// TIA Portal project "DT_PSA_OPCV" (V19)

(* hardware
DEVICE "S7-1500/ET200MP-Station_1"  S7-1500 station
   slot 0: "Profilschiene_0"  Rack  6ES7 590-1***0-0AA0
   slot 1: "PLC_1"  CPU 1516F-3 PN/DP  6ES7 516-3FN02-0AB0  V2.9
      slot 3: "CPU-Display_1"  6ES7591-1BA00-0AA0
      slot 32768: "PROFINET-Schnittstelle_1"  X1
         slot 32769: "Port_1"  X1 P1
         slot 32770: "Port_2"  X1 P2
      slot 33024: "PROFINET-Schnittstelle_2"  X2
         slot 33025: "Port_1"  X2 P1
      slot 33280: "DP-Schnittstelle_1"  X3
      slot 34817: "Virtual CP interface port_1"  Virtual CP interface port  Virtual CP interface port
   slot 2: "DI 16x24VDC HF_1"  DI 16x24VDC HF  6ES7 521-1BH00-0AB0  V2.2
   slot 3: "DQ 8x24VDC/2A HF_1"  DQ 8x24VDC/2A HF  6ES7 522-1BF00-0AB0  V2.2
   slot 4: "F-DI 16x24V DC_1"  F-DI 16x24V DC  6ES7 526-1BH00-0AB0  V1.0
      slot 1: "F-DI 16x24V DC_1"  F-DI 16x24V DC
   slot 5: "F-DQ 8x24V DC/2A PPM_1"  F-DQ 8x24V DC/2A PPM  6ES7 526-2BF00-0AB0  V1.0
      slot 1: "F-DQ 8x24V DC/2A PPM_1"  F-DQ 8x24V DC/2A PPM
DEVICE "HMI_1"  TP700 Comfort
   slot 0: "HMI_1"  TP700 Comfort  6AV2 124-0GC01-0AX0  17.0.0.0
   slot 1: "HMI_RT_1"  TP700 Comfort  6AV2 124-0GC01-0AX0  17.0.0.0
   slot 5: "HMI_1.IE_CP_1"  PROFINET Interface  17.0.0.0
      slot 1: "PROFINET Schnittstelle_1"  PROFINET Interface
         slot 1: "Port_1"  Port
         slot 2: "Port_2"  Port
   slot 7: "HMI_1.MPI/DP_CP_1"  MPI/DP Interface  17.0.0.0
*)

// ===== PLC "PLC_1"  CPU 1516F-3 PN/DP =====
// protected blocks, not shown: "Main_Safety_RTG1", "Main_Safety_RTG1_DB"

VAR_GLOBAL   // PLC tag table "Control Panel"
   "BT2_OpMode" AT %I0.2 : Bool;   // Betriebsart: 1=Automatik / 0=Hand
   "BT3_SingleStep" AT %I0.3 : Bool;   // Einzelschritt ausführen
   "BT4_AutoStart" AT %I0.4 : Bool;   // Automatik Ein
   "BT5_AutoStop" AT %I0.5 : Bool;   // Automatik Halt
   "BT7_Reset" AT %I0.7 : Bool;   // Grundstellung
   "BT6_Ack" AT %I0.6 : Bool;   // Störung quittieren
   "BT1_ControlLight" AT %Q0.1 : Bool;   // Tasterbeleuchtung "Steuerung läuft" (grün)
   "BT4_AutoLight" AT %Q0.4 : Bool;   // Tasterbeleuchtung "Automatik läuft" (grün)
   "BT6_ErrFltLight" AT %Q0.6 : Bool;   // Tasterbeleuchtung "Lampe Störung" (rot)
   "SignalTower_Yellow" AT %Q1.2 : Bool;   // Ampel "Lampe Einrichten aktiv" (gelb)
   "BT1_ControlOnOff" AT %I0.1 : Bool;   // 1 = Steuerung Ein (einrastend)
   "SignalTower_Green" AT %Q1.1 : Bool;   // Ampel "Automatik läuft" (grün)
   "SignalTower_Red" AT %Q1.3 : Bool;   // Ampel "Störung" (rot)
   "BT3_SingleStepLight" AT %Q0.3 : Bool;   // Tasterbeleuchtung "Einzelschritt läuft" (grün)
   "BT7_HomingLight" AT %Q0.7 : Bool;   // Tasterbeleuchtung "Grundstellungsfahrt läuft" (green)
   "BT5_AutoStopLight" AT %Q0.5 : Bool;   // Tasterbeleuchtung "Automatik Stop läuft" (blau)
   "BT8_ImmediateStop" AT %I1.0 : Bool;   // Sofort Halt
   "BT8_ImmediateStopLight" AT %Q1.0 : Bool;   // Tasterbeleuchtung "Sofort Halt" (rot)
END_VAR

VAR_GLOBAL   // PLC tag table "System"
   "Clock_Byte" AT %MB0 : Byte;
   "Clock_10Hz" AT %M0.0 : Bool;
   "Clock_5Hz" AT %M0.1 : Bool;
   "Clock_2.5Hz" AT %M0.2 : Bool;
   "Clock_2Hz" AT %M0.3 : Bool;
   "Clock_1.25Hz" AT %M0.4 : Bool;
   "Clock_1Hz" AT %M0.5 : Bool;
   "Clock_0.625Hz" AT %M0.6 : Bool;
   "Clock_0.5Hz" AT %M0.7 : Bool;
   "System_Byte" AT %MB1 : Byte;
   "FirstScan" AT %M1.0 : Bool;
   "DiagStatusUpdate" AT %M1.1 : Bool;
   "AlwaysTRUE" AT %M1.2 : Bool;
   "AlwaysFALSE" AT %M1.3 : Bool;
   "Commissioning_True" AT %M2.0 : Bool;
END_VAR

VAR_GLOBAL CONSTANT   // PLC tag table "System"
   "SYS_MACHINE_MAXSTATIONS" : USInt := 10;   // Anzahl Stationen pro Maschine
   "SYS_SQ_MAXSEQUENCES" : USInt := 12;   // Anzahl Schrittketten pro Station
   "SYS_DRIVE_POSITIONS" : USInt := 8;   // Anzahl Positionen pro Servoantrieb
   "SYS_MANUALMOVEMENTS" : UInt := 64;   // Anzahl maximaler Einrichtfunktionen
   "SYS_HMI_SETUPMAXROWS" : USInt := 6;   // HMI Vorgabe maximale Anzahl an Einrichtzeilen auf der Steuerung verfügbar
END_VAR

VAR_GLOBAL   // PLC tag table "FG01"
   "FG01_Y_Gripper_InHome" AT %I101.0 : Bool;   // geöffnet
   "FG01_Y_Gripper_InWork" AT %I101.1 : Bool;   // geschlossen
   "FG01_Y_Gripper_WorkPos" AT %Q101.1 : Bool;   // schließen
   "FG01_Y_Plattform_InHome" AT %I102.0 : Bool;   // hinten
   "FG01_Y_Plattform_InWork" AT %I102.1 : Bool;   // vorne
   "FG01_Y_Plattform_HomePos" AT %Q102.0 : Bool;
   "FG01_Y_Plattform_WorkPos" AT %Q102.1 : Bool;
   "FG01_Y_ReaderWindow_InWork" AT %I103.1 : Bool;
   "FG01_Y_ReaderWindow_WorkPos" AT %Q103.1 : Bool;   // Position zum Code Lesen
   "FG01_Y_Gripper_HomePos" AT %Q101.0 : Bool;   // öffnen
   "FG01_Y_ReaderWindow_HomePos" AT %Q103.0 : Bool;
END_VAR

VAR_GLOBAL   // PLC tag table "FG03"
   "FG03_Y_AxisR1_InHome" AT %I301.0 : Bool;
   "FG03_Y_AxisR1_InWork" AT %I301.1 : Bool;
   "FG03_Y_AxisR1_HomePos" AT %Q301.0 : Bool;
   "FG03_Y_AxisR1_WorkPos" AT %Q301.1 : Bool;
   "FG03_Y_AxisX1_InHome" AT %I302.0 : Bool;
   "FG03_Y_AxisX1_InWork" AT %I302.1 : Bool;
   "FG03_Y_AxisX1_HomePos" AT %Q302.0 : Bool;
   "FG03_Y_AxisX1_WorkPos" AT %Q302.1 : Bool;
   "FG03_Y_AxisY1_InHome" AT %I303.0 : Bool;
   "FG03_Y_AxisY1_InWork" AT %I303.1 : Bool;
   "FG03_Y_AxisY1_HomePos" AT %Q303.0 : Bool;
   "FG03_Y_AxisY1_WorkPos" AT %Q303.1 : Bool;
   "FG03_Y_AxisX2_InHome" AT %I304.0 : Bool;
   "FG03_Y_AxisX2_InWork" AT %I304.1 : Bool;
   "FG03_Y_AxisX2_HomePos" AT %Q304.0 : Bool;
   "FG03_Y_AxisX2_WorkPos" AT %Q304.1 : Bool;
   "FG03_Y_AxisY2_InHome" AT %I305.0 : Bool;
   "FG03_Y_AxisY2_InWork" AT %I305.1 : Bool;
   "FG03_Y_AxisY2_HomePos" AT %Q305.0 : Bool;
   "FG03_Y_AxisY2_WorkPos" AT %Q305.1 : Bool;
   "FG03_Y_Gripper1_InHome" AT %I306.0 : Bool;
   "FG03_Y_Gripper1_InWork" AT %I306.1 : Bool;
   "FG03_Y_Gripper1_HomePos" AT %Q306.0 : Bool;
   "FG03_Y_Gripper1_WorkPos" AT %Q306.1 : Bool;
   "FG03_Y_Gripper2_InHome" AT %I307.0 : Bool;
   "FG03_Y_Gripper2_InWork" AT %I307.1 : Bool;
   "FG03_Y_Gripper2_HomePos" AT %Q307.0 : Bool;
   "FG03_Y_Gripper2_WorkPos" AT %Q307.1 : Bool;
END_VAR

VAR_GLOBAL   // PLC tag table "FG04"
   "FG04_Y_AxisZ_InWork" AT %I401.1 : Bool;
   "FG04_Y_AxisZ_WorkPos" AT %Q401.1 : Bool;
   "FG04_Y_AxisZ_HomePos" AT %Q401.0 : Bool;
   "FG04_Y_AxisZ_InHome" AT %I401.0 : Bool;
END_VAR

VAR_GLOBAL   // PLC tag table "FG05"
   "FG05_B_Part" AT %I500.0 : Bool;
   "FG05_Y_AxisR_InHome" AT %I501.0 : Bool;
   "FG05_Y_AxisR_InWork" AT %I501.1 : Bool;
   "FG05_Y_AxisR_HomePos" AT %Q501.0 : Bool;
   "FG05_Y_AxisR_WorkPos" AT %Q501.1 : Bool;
   "FG05_Y_AxisX_InHome" AT %I502.0 : Bool;
   "FG05_Y_AxisX_InWork" AT %I502.1 : Bool;
   "FG05_Y_AxisX_HomePos" AT %Q502.0 : Bool;
   "FG05_Y_AxisX_WorkPos" AT %Q502.1 : Bool;
   "FG05_Y_AxisZ1_InHome" AT %I503.0 : Bool;
   "FG05_Y_AxisZ1_InWork" AT %I503.1 : Bool;
   "FG05_Y_AxisZ1_HomePos" AT %Q503.0 : Bool;
   "FG05_Y_AxisZ1_WorkPos" AT %Q503.1 : Bool;
   "FG05_Y_AxisZ2_InHome" AT %I504.0 : Bool;
   "FG05_Y_AxisZ2_InWork" AT %I504.1 : Bool;
   "FG05_Y_AxisZ2_HomePos" AT %Q504.0 : Bool;
   "FG05_Y_AxisZ2_WorkPos" AT %Q504.1 : Bool;
   "FG05_Y_CapsSourceStopper_InHome" AT %I505.0 : Bool;   // GS = Kaps können vereinzelt werden
   "FG05_Y_CapsSourceStopper_WorkPos" AT %Q505.1 : Bool;   // AS = Vereinzelung kann geleert werden (Vereinzelung nicht möglich)
   "FG05_Y_Gripper_InHome" AT %I506.0 : Bool;
   "FG05_Y_Gripper_InWork" AT %I506.1 : Bool;
   "FG05_Y_Gripper_HomePos" AT %Q506.0 : Bool;
   "FG05_Y_Gripper_WorkPos" AT %Q506.1 : Bool;
   "FG05_Y_CapsSourceStopper_HomePos" AT %Q505.0 : Bool;
   "FG05_M_Bunker" AT %Q507.0 : Bool;   // Sortiertopf ein
   "FG05_M_Conveyor" AT %Q507.1 : Bool;   // Linearförderer ein
END_VAR

VAR_GLOBAL   // PLC tag table "FG_Transport"
   "FG_TS_Gate_1_InHome" AT %I1001.0 : Bool;   // geöffnet
   "FG_TS_Gate_1_InWork" AT %I1001.1 : Bool;   // geschlossen
   "FG_TS_Gate_1_WorkPos" AT %Q1001.1 : Bool;   // Schließen
   "FG_TS_Gate_2_InHome" AT %I1002.0 : Bool;   // geöffnet
   "FG_TS_Gate_2_InWork" AT %I1002.1 : Bool;   // geschlossen
   "FG_TS_Gate_2_WorkPos" AT %Q1002.1 : Bool;   // Schließen
   "FG_TS_Index01_B_Detect" AT %I1003.0 : Bool;   // 1 = erkannt
   "FG_TS_Index01_B_Exit" AT %I1003.1 : Bool;   // 1 = erkannt
   "FG_TS_Index01_Y_Lift_InHome" AT %I1003.2 : Bool;   // Heber ist unten
   "FG_TS_Index01_Y_Lift_InWork" AT %I1003.3 : Bool;   // Heber ist oben
   "FG_TS_Index01_Y_Lift_HomePos" AT %Q1003.0 : Bool;   // Heber senken
   "FG_TS_Index01_Y_Lift_WorkPos" AT %Q1003.1 : Bool;   // Heber heben
   "FG_TS_Index01_Y_Stopper_InHome" AT %I1003.4 : Bool;   // Stopper geschlossen
   "FG_TS_Index01_Y_Stopper_WorkPos" AT %Q1003.2 : Bool;   // Stopper öffnen
   "FG_TS_Index02_B_Detect" AT %I1004.0 : Bool;   // 1 = erkannt
   "FG_TS_Index02_B_Exit" AT %I1004.1 : Bool;   // 1 = erkannt
   "FG_TS_Index02_Y_Lift_InHome" AT %I1004.2 : Bool;   // Heber ist unten
   "FG_TS_Index02_Y_Lift_InWork" AT %I1004.3 : Bool;   // Heber ist oben
   "FG_TS_Index02_Y_Lift_HomePos" AT %Q1004.0 : Bool;   // Heber senken
   "FG_TS_Index02_Y_Lift_WorkPos" AT %Q1004.1 : Bool;   // Heber heben
   "FG_TS_Index02_Y_Stopper_InHome" AT %I1004.4 : Bool;   // Stopper geschlossen
   "FG_TS_Index02_Y_Stopper_WorkPos" AT %Q1004.2 : Bool;   // Stopper öffnen
   "FG_TS_Index03_B_Detect" AT %I1005.0 : Bool;   // 1 = erkannt
   "FG_TS_Index03_B_Exit" AT %I1005.1 : Bool;   // 1 = erkannt
   "FG_TS_Index03_Y_Lift_InHome" AT %I1005.2 : Bool;   // Heber ist unten
   "FG_TS_Index03_Y_Lift_InWork" AT %I1005.3 : Bool;   // Heber ist oben
   "FG_TS_Index03_Y_Lift_HomePos" AT %Q1005.0 : Bool;   // Heber senken
   "FG_TS_Index03_Y_Lift_WorkPos" AT %Q1005.1 : Bool;   // Heber heben
   "FG_TS_Index03_Y_Stopper_InHome" AT %I1005.4 : Bool;   // Stopper geschlossen
   "FG_TS_Index03_Y_Stopper_WorkPos" AT %Q1005.2 : Bool;   // Stopper öffnen
   "FG_TS_Index04_B_Detect" AT %I1006.0 : Bool;   // 1 = erkannt
   "FG_TS_Index04_B_Exit" AT %I1006.1 : Bool;   // 1 = erkannt
   "FG_TS_Index04_Y_Lift_InHome" AT %I1006.2 : Bool;   // Heber ist unten
   "FG_TS_Index04_Y_Lift_InWork" AT %I1006.3 : Bool;   // Heber ist oben
   "FG_TS_Index04_Y_Lift_HomePos" AT %Q1006.0 : Bool;   // Heber senken
   "FG_TS_Index04_Y_Lift_WorkPos" AT %Q1006.1 : Bool;   // Heber heben
   "FG_TS_Index04_Y_Stopper_InHome" AT %I1006.4 : Bool;   // Stopper geschlossen
   "FG_TS_Index04_Y_Stopper_WorkPos" AT %Q1006.2 : Bool;   // Stopper öffnen
   "FG_TS_Index05_B_Detect" AT %I1007.0 : Bool;   // 1 = erkannt
   "FG_TS_Index05_B_Exit" AT %I1007.1 : Bool;   // 1 = erkannt
   "FG_TS_Index05_Y_Lift_InHome" AT %I1007.2 : Bool;   // Heber ist unten
   "FG_TS_Index05_Y_Lift_InWork" AT %I1007.3 : Bool;   // Heber ist oben
   "FG_TS_Index05_Y_Lift_HomePos" AT %Q1007.0 : Bool;   // Heber senken
   "FG_TS_Index05_Y_Lift_WorkPos" AT %Q1007.1 : Bool;   // Heber heben
   "FG_TS_Index05_Y_Stopper_InHome" AT %I1007.4 : Bool;   // Stopper geschlossen
   "FG_TS_Index05_Y_Stopper_WorkPos" AT %Q1007.2 : Bool;   // Stopper öffnen
   "FG_TS_Stopper01_B_Detect" AT %I1008.0 : Bool;   // 1 = erkannt
   "FG_TS_Stopper01_B_Exit" AT %I1008.1 : Bool;   // 1 = erkannt
   "FG_TS_Stopper01_Y_Stopper_InHome" AT %I1008.4 : Bool;   // Stopper geschlossen
   "FG_TS_Stopper01_Y_Stopper_WorkPos" AT %Q1008.2 : Bool;   // Stopper öffnen
   "FG_TS_Stopper02_B_Detect" AT %I1009.0 : Bool;   // 1 = erkannt
   "FG_TS_Stopper02_B_Exit" AT %I1009.1 : Bool;   // 1 = erkannt
   "FG_TS_Stopper02_Y_Stopper_InHome" AT %I1009.4 : Bool;   // Stopper geschlossen
   "FG_TS_Stopper02_Y_Stopper_WorkPos" AT %Q1009.2 : Bool;   // Stopper öffnen
   "FG_TS_Stopper03_B_Detect" AT %I1010.0 : Bool;   // 1 = erkannt
   "FG_TS_Stopper03_B_Exit" AT %I1010.1 : Bool;   // 1 = erkannt
   "FG_TS_Stopper03_Y_Stopper_InHome" AT %I1010.4 : Bool;   // Stopper geschlossen
   "FG_TS_Stopper03_Y_Stopper_WorkPos" AT %Q1010.2 : Bool;   // Stopper öffnen
   "FG_TS_Stopper04_B_Detect" AT %I1011.0 : Bool;   // 1 = erkannt
   "FG_TS_Stopper04_B_Exit" AT %I1011.1 : Bool;   // 1 = erkannt
   "FG_TS_Stopper04_Y_Stopper_InHome" AT %I1011.4 : Bool;   // Stopper geschlossen
   "FG_TS_Stopper04_Y_Stopper_WorkPos" AT %Q1011.2 : Bool;   // Stopper öffnen
   "FG_TS_Lift01_B_Detect" AT %I1012.0 : Bool;   // 1 = erkannt
   "FG_TS_Lift01_B_Exit" AT %I1012.1 : Bool;   // 1 = erkannt
   "FG_TS_Lift01_Y_Lift_InHome" AT %I1012.2 : Bool;   // Heber ist unten
   "FG_TS_Lift01_Y_Lift_InWork" AT %I1012.3 : Bool;   // Heber ist oben
   "FG_TS_Lift01_Y_Lift_HomePos" AT %Q1012.0 : Bool;   // Heber senken
   "FG_TS_Lift01_Y_Lift_WorkPos" AT %Q1012.1 : Bool;   // Heber heben
   "FG_TS_Lift01_M_Conveyor_Plus" AT %Q1012.2 : Bool;   // Antrieb vorwärts
   "FG_TS_Lift01_M_Conveyor_Minus" AT %Q1012.3 : Bool;   // Antrieb rückwärts
   "FG_TS_Lift02_B_Detect" AT %I1013.0 : Bool;   // 1 = erkannt
   "FG_TS_Lift02_B_Exit" AT %I1013.1 : Bool;   // 1 = erkannt
   "FG_TS_Lift02_Y_Lift_InHome" AT %I1013.2 : Bool;   // Heber ist unten
   "FG_TS_Lift02_Y_Lift_InWork" AT %I1013.3 : Bool;   // Heber ist oben
   "FG_TS_Lift02_Y_Lift_HomePos" AT %Q1013.0 : Bool;   // Heber senken
   "FG_TS_Lift02_Y_Lift_WorkPos" AT %Q1013.1 : Bool;   // Heber heben
   "FG_TS_Lift02_M_Conveyor_Plus" AT %Q1013.2 : Bool;   // Antrieb vorwärts
   "FG_TS_Lift02_M_Conveyor_Minus" AT %Q1013.3 : Bool;   // Antrieb rückwärts
   "FG_TS_Transport01_M_Conveyor_Plus" AT %Q1014.0 : Bool;   // Antrieb vorwärts
   "FG_TS_Transport01_M_Conveyor_Minus" AT %Q1014.1 : Bool;   // Antrieb rückwärts
   "FG_TS_Transport02_M_Conveyor_Plus" AT %Q1015.0 : Bool;   // Antrieb vorwärts
   "FG_TS_Transport02_M_Conveyor_Minus" AT %Q1015.1 : Bool;   // Antrieb rückwärts
END_VAR

VAR_GLOBAL   // PLC tag table "Safety"
   "i_SS_ESTOP1" AT %I50.0 : Bool;
   "q_SS_ESTOP1" AT %Q50.0 : Bool;
END_VAR

// folder: Actors/ActorTypes

TYPE "typeActor"
   STRUCT
      setHomePos : Bool;   // Grundstellung ansteuern
      setWorkPos : Bool;   // Arbeitsstellung ansteuern
      inHomePos : Bool;   // steht in Grundstellung
      inWorkPos : Bool;   // steht in Arbeitsstellung
      homeAct : Bool;   // Grundstellung wird angesteuert
      workAct : Bool;   // Arbeitsstellung wird angesteuert
      homeIsInterlocked : Bool;   // 1 = Grundstellung ist gesperrt
      workIsInterlocked : Bool;   // 1 = Arbeitsstellung ist gesperrt
   END_STRUCT;
END_TYPE

TYPE "typeActor_2Out0In"
   STRUCT
      setHomePos : Bool;   // Grundstellung ansteuern
      setWorkPos : Bool;   // Arbeitsstellung ansteuern
      homeAct : Bool;   // Grundstellung wird angesteuert
      workAct : Bool;   // Arbeitsstellung wird angesteuert
      homeIsInterlocked : Bool;   // 1 = Grundstellung ist gesperrt
      workIsInterlocked : Bool;   // 1 = Arbeitsstellung ist gesperrt
      setError : Bool;   // in Störung setzen
      inError : Bool;   // Störung vorhanden
   END_STRUCT;
END_TYPE

TYPE "typeActor_2Out2In"
   STRUCT
      setHomePos : Bool;   // Grundstellung ansteuern
      setWorkPos : Bool;   // Arbeitsstellung ansteuern
      inHomePos : Bool;   // steht in Grundstellung
      inWorkPos : Bool;   // steht in Arbeitsstellung
      homeAct : Bool;   // Grundstellung wird angesteuert
      workAct : Bool;   // Arbeitsstellung wird angesteuert
      homeIsInterlocked : Bool;   // 1 = Grundstellung ist gesperrt
      workIsInterlocked : Bool;   // 1 = Arbeitsstellung ist gesperrt
      setError : Bool;   // in Störung setzen
      inError : Bool;   // Störung vorhanden
   END_STRUCT;
END_TYPE

TYPE "typeActor_1Out0In"
   STRUCT
      setWorkPos : Bool;   // Arbeitsstellung ansteuern
      workAct : Bool;   // Arbeitsstellung wird angesteuert
      workIsInterlocked : Bool;   // 1 = Arbeitsstellung ist gesperrt
      setError : Bool;   // in Störung setzen
      inError : Bool;   // Störung vorhanden
   END_STRUCT;
END_TYPE

TYPE "typeActor_1Out2In"
   STRUCT
      setWorkPos : Bool;   // Arbeitsstellung ansteuern
      inHomePos : Bool;   // steht in Grundstellung
      inWorkPos : Bool;   // steht in Arbeitsstellung
      workAct : Bool;   // Arbeitsstellung wird angesteuert
      workIsInterlocked : Bool;   // 1 = Arbeitsstellung ist gesperrt
      setError : Bool;   // in Störung setzen
      inError : Bool;   // Störung vorhanden
   END_STRUCT;
END_TYPE

TYPE "typeActor_2Out1In"
   STRUCT
      setHomePos : Bool;   // Grundstellung ansteuern
      setWorkPos : Bool;   // Arbeitsstellung ansteuern
      inHomePos : Bool;   // steht in Grundstellung
      inWorkPos : Bool;   // steht in Arbeitsstellung
      homeAct : Bool;   // Grundstellung wird angesteuert
      workAct : Bool;   // Arbeitsstellung wird angesteuert
      homeIsInterlocked : Bool;   // 1 = Grundstellung ist gesperrt
      workIsInterlocked : Bool;   // 1 = Arbeitsstellung ist gesperrt
      setError : Bool;   // in Störung setzen
      inError : Bool;   // Störung vorhanden
   END_STRUCT;
END_TYPE

TYPE "typeActor_1Out1In"
   STRUCT
      setWorkPos : Bool;   // Arbeitsstellung ansteuern
      inHomePos : Bool;   // steht in Grundstellung
      inWorkPos : Bool;   // steht in Arbeitsstellung
      workAct : Bool;   // Arbeitsstellung wird angesteuert
      workIsInterlocked : Bool;   // 1 = Arbeitsstellung ist gesperrt
      setError : Bool;   // in Störung setzen
      inError : Bool;   // Störung vorhanden
   END_STRUCT;
END_TYPE

// folder: Actors/Drives

TYPE "typeDriveData"
   STRUCT
      position : Array[1.."SYS_DRIVE_POSITIONS"] of Real;   // Positionsvorgabe
      speed : Array[1.."SYS_DRIVE_POSITIONS"] of Real;   // Geschwindigkeitsvorgabe
   END_STRUCT;
   // // position[1] : Grundstellung (reserviert)
END_TYPE

TYPE "typeDriveControl"
   STRUCT
      moveToPos : Array[1.."SYS_DRIVE_POSITIONS"] of Bool;   // Fahrbefehl ausführen
      jog : Struct   // Handbetrieb
         pos : Bool;   // Tippen positiv
         neg : Bool;   // Tippen negativ
         "step" : Real;   // Tippschrittweite
         speed : Real;   // Tippgeschwindigkeit
      END_STRUCT;
   END_STRUCT;
END_TYPE

TYPE "typeDriveStatus"
   STRUCT
      ready : Bool;   // Bereit
      error : Bool;   // Störung
      posReached : Bool;   // Positionsvorgabe erreicht
      actualPosition : Real;   // Ist-Position
      actualSpeed : Real;   // Ist-Geschwindigkeit
      interlockMin : Bool;   // 1 = Fahrtrichtung zur Endposition min gesperrt
      interlockMax : Bool;   // 1 = Fahrtrichtung zur Endposition max gesperrt
      endPosMin : Bool;   // Endposition min erreicht
      endPosMax : Bool;   // Endposition max erreicht
      inHomePos : Bool;   // steht in Grundstellung
   END_STRUCT;
END_TYPE

TYPE "typeDriveConverter"
   STRUCT
      actualPosition : Real;   // Ist-Position (Drive-Einheit)
      actualSpeed : Real;   // Ist-Geschwindigkeit (Drive-Einheit)
      setPosition : Real;   // Sollposition (Drive-Einheit)
      setSpeed : Real;   // Sollgeschwindigkeit (Drive-Einheit)
      minPosDrive : Real;   // Minimale Positionierung (Drive-Einheit)
      maxPosDrive : Real;   // Maximale Positionierung (Drive-Einheit)
      maxSpeedDrive : Real;   // Maximale Geschwindigkeit (Drive-Einheit)
      posOffset : Real;   // Offset für Positionsfensterfreigabe (Drive-Einheit)
      ready : Bool;   // Umrichter Bereit
      error : Bool;   // Umrichter Störung
      posReached : Bool;   // Position erreicht
      releaseMotion : Bool;   // Bewegungsfreigabe
   END_STRUCT;
END_TYPE

// folder: HMI/Errors_Messages

TYPE "typePlcErrors"
   STRUCT
      errorNo : Array[1..64] of Bool;
   END_STRUCT;
END_TYPE

TYPE "typeHmiErrMsg"
   STRUCT
      message : Array[1..2] of Word;   // Meldung auslösen
      alarmAckPlc : Array[1..8] of Word;   // Fehler auslösen und Quittierung über SPS
      ackHmi : Array[1..4] of Word;   // Quittierung über HMI
   END_STRUCT;
END_TYPE

TYPE "typePlcErrMsg"
   STRUCT
      messages : "typePlcMessages";
      alarms : "typePlcErrors";
   END_STRUCT;
END_TYPE

TYPE "typePlcMessages"
   STRUCT
      msgNo : Array[1..32] of Bool;
   END_STRUCT;
END_TYPE

// folder: HMI/ManualMovement

TYPE "typeHmiManualMove"
   STRUCT
      move : "typeManualMove";   // Bewegung
      movementNo : USInt;   // Nummer der Bewegungsfunktion
      textlistFunctionName : UInt;   // Funktionsname: Wert für Textliste
      textlistFunctionExecuteLeft : UInt;   // Bewegung Links: Wert für Textliste
      textlistFunctionFinalPosLeft : UInt;   // Endposition Links: Wert für Textliste
      textlistFunctionExecuteRight : UInt;   // Bewegung Rechts: Wert für Textliste
      textlistFunctionFinalPosRight : UInt;   // Endposition Rechts: Wert für Textliste
   END_STRUCT;
END_TYPE

TYPE "typeHmiManualMovement"
   STRUCT
      selection : Struct
         station : USInt;   // Angewählte Station
         page : USInt;   // Aktuele Seite
         ofMaxPages : USInt;   // von maximal Seiten
         nextPage : Bool;   // Schaltfläche: Nächste Seite
         previousPage : Bool;   // Schaltfläche: Vorherige Seite
         showSymbols : Bool;   // Schaltfläche: Zeige symbolische Ansicht
      END_STRUCT;
      rows : Array[1.."SYS_HMI_SETUPMAXROWS"] of "typeHmiManualMove";
   END_STRUCT;
END_TYPE

// folder: Machine

TYPE "typeMachine"
   STRUCT
      controlOn : Bool;   // Maschinensteuerung ist eingeschaltet
      automaticMode : Bool;   // Betriebsart Automatik ist aktiv
      automaticIsRunning : Bool;   // Automatik (bzw. ReleaseCycle) läuft in mindestens einer Station
      automaticStart : Bool;   // Automatikstart auslösen
      automaticStops : Bool;   // Automatik stoppt
      singleStepPulse : Bool;   // Einzelschritt
      immediateStop : Bool;   // Sofort Halt der Stationen auslösen
      acknowledge : Bool;   // Quittierung
      reset : Bool;   // Neustart/Grundstellung auslösen
      isInError : Bool;   // Störung vorhanden
      isHoming : Bool;   // Maschinengrundstellungsfahrt wird ausgeführt
      isInHome : Bool;   // Alle Stationen sind in Grundstellung
   END_STRUCT;
END_TYPE

TYPE "typeStation"
   STRUCT
      exists : Bool := false;   // true = Station existiert / false = Platzhalter
      signals : "typeStationSignals";
      stepSeqs : "typeStepSequences";
   END_STRUCT;
END_TYPE

TYPE "typeStations"
   STRUCT
      station : Array[1.."SYS_MACHINE_MAXSTATIONS"] of "typeStation";
   END_STRUCT;
END_TYPE

TYPE "typeStepSequence"
   STRUCT
      exists : Bool;   // Schrittkette verfügbar
      start : Bool;   // Start Schrittkette
      running : Bool;   // Schrittkette läuft
      done : Bool;   // Schrittkette ist fertig
      error : Bool;   // Störung vorhanden
      init : Bool;   // Initialschritt aktiv
      inHome : Bool;   // Steht in Grundstellung
      isWaiting : Bool;   // Steht im Warteschritt
      inHoming : Bool;   // Grundstellungsfahrt aktiv
      jogDone : Bool;   // Halbautomatische Weiterschaltung abgeschlossen
   END_STRUCT;
END_TYPE

TYPE "typeStepSequences"
   STRUCT
      stepSeq : Array[1.."SYS_SQ_MAXSEQUENCES"] of "typeStepSequence";   // Schrittkette
   END_STRUCT;
END_TYPE

TYPE "typeMachineSafety"
   STRUCT
      EStopOk : Bool;   // Not-Aus Kreis ok
      RunUpPneumatic : Bool;
      PneumaticIsOk : Bool;
      Error : Bool;
   END_STRUCT;
END_TYPE

TYPE "typeStationSignals"
   STRUCT
      safetyOk : Bool;   // Sicherheit ist ok
      controlOn : Bool;   // Steuerung eingeschaltet
      automaticMode : Bool;   // Automatikmodus angewählt
      modeSetup : Bool;   // Handmodus angewählt
      modeAuto : Bool;   // Betriebsart: Automatik aktiv
      modeTap : Bool;   // Betriebsart: Einzelschritt aktiv
      releaseCycle : Bool;   // Bearbeitungsfreigabe
      releaseNextJog : Bool;   // Freigabe Weiterschaltung (Zünd-Impuls für Schrittketten)
      resetCycle : Bool;   // Ablauf neustarten
      setupActive : Bool;   // Handmodus/Einrichten aktiv (mindestens 1 Aktor ist in Hand bewegt worden)
      ack : Bool;   // Quittieren
      singlePulse : Bool;   // Einzelschritt auslösen
      autoIsStoping : Bool;   // Automatikstopp/Zyklusende angewählt
      isStopped : Bool;   // Automatikabläufe/Graphen sind angehalten
      isHoming : Bool;   // Grundstellungsablauf aktiv
      isInHome : Bool;   // steht in Grundstellung
      isInError : Bool;   // Störung vorhanden
      actorError : Bool;   // Mindestens ein Stationsaktor hat eine Störung (wird in Aktor-Bausteinen gesetzt)
   END_STRUCT;
END_TYPE

// folder: Machine/ManualMovement

TYPE "typeManualMove"
   STRUCT
      control : "typeManualMoveControl";   // Steuerung
      attributes : "typeManualMoveAttributes";   // Eigenschaften
   END_STRUCT;
END_TYPE

TYPE "typeManualMoveSetup"
   STRUCT
      initialisation : Struct   // Für den Initialisierungsdurchlauf notwendig
         execute : Bool;   // Initialisierung der Bewegungsfunktionen ausführen
         isActive : Bool;   // Initialisierung läuft
         isDone : Bool;   // Initialisierung abgeschlossen
         error : Bool;   // Initialisierung fehlerhaft
         currentStationNo : USInt;   // Hilfsspeicher für die Station
         currentMoveNo : USInt;   // Hilfsspeicher für die Bewegungsnummer innerhalb der Station
         moveNo : USInt;   // Hilfsspeicher für die Bewegungsnummer (maximale Anzahl Stationen wenn initalisiert)
      END_STRUCT;
   END_STRUCT;
END_TYPE

TYPE "typeManualMovements"
   STRUCT
      setup : "typeManualMoveSetup";
      movements : Array[0.."SYS_MANUALMOVEMENTS"] of "typeManualMove";
   END_STRUCT;
   // // movements[0] : not useable
END_TYPE

TYPE "typeManualMoveControl"
   STRUCT
      moveHomePos : Bool;   // Grundstellung ansteuern
      moveWorkPos : Bool;   // Arbeitsstellung ansteuern
      inHomePos : Bool;   // steht in Grundstellung
      inWorkPos : Bool;   // steht in Arbeitsstellung
      homeAct : Bool;   // Grundstellung wird angesteuert
      workAct : Bool;   // Arbeitsstellung wird angesteuert
      homeIsInterlocked : Bool;   // 1 = Grundstellung ist gesperrt
      workIsInterlocked : Bool;   // 1 = Arbeitsstellung ist gesperrt
      value : Real;   // Dezimalanzeige
   END_STRUCT;
END_TYPE

TYPE "typeManualMoveAttributes"
   STRUCT
      initialised : Bool;   // Ist initialisiert
      showValue : Bool;   // Zeige Dezimalanzeige
      showName : Bool;   // Zeige Benennung der Einrichtzeile
      showRecRight : Bool;   // Zeige Rechteck Rechts
      showRecLeft : Bool;   // Zeige Rechteck Links
      isExecutableRight : Bool;   // Ist ausführbar rechte Seite
      isExecutableLeft : Bool;   // Ist ausführbar linke Seite
      hasEndPositionRight : Bool;   // Zeige Endposition rechte Seite
      hasEndPositionLeft : Bool;   // Zeige Endposition linke Seite
      stationNo : USInt;   // Zugehörige Stationsnummer
      movementNo : USInt;   // Zugehörige Bewegungsnummer innerhalb der Station
   END_STRUCT;
END_TYPE

// folder: Simulation

TYPE "typeSimInterface"
   STRUCT
      Simulation : Bool;   // Simulation vorhanden
      SimulationStandalone : Bool;   // Nur virtuelle Maschine vorhanden
      Started : Bool;   // Simulation wurde gestartet (SPS-Eingang)
      Synchronized : Bool;   // Simulation und SPS sind synchronisiert (SPS-Ausgang)
   END_STRUCT;
END_TYPE

TYPE "typeSimAktor2Ins2Outs"
   STRUCT
      ixHomePos : Bool;   // Simulation ist in Grundstellung
      ixWorkPos : Bool;   // Simulation ist in Arbeitsstellung
      qxSetHomePos : Bool;   // Setze Grundstellung in der Simulation
      qxSetWorkPos : Bool;   // Setze Arbeitsstellung in der Simulation
      "0_4" : Bool;
      "0_5" : Bool;
      "0_6" : Bool;
      "0_7" : Bool;
   END_STRUCT;
END_TYPE

// folder: 1. HMI

DATA_BLOCK "InstHmiManualMovementController"   // DB1003
{ S7_Optimized_Access := 'TRUE' }
VERSION : 0.1
// stored: InstanceOfName HmiManualMovementController
"HmiManualMovementController"
BEGIN
END_DATA_BLOCK

DATA_BLOCK "HmiManualMovement"   // DB1004
{ S7_Optimized_Access := 'TRUE' }
VERSION : 0.1
BEGIN
END_DATA_BLOCK

// folder: 10_Simulation (unused)

DATA_BLOCK "SimulationInterface"   // DB9
{ S7_Optimized_Access := 'TRUE' }
VERSION : 0.1
   VAR
      Interface : "typeSimInterface";
   END_VAR
BEGIN
   Interface.Simulation := 1;
END_DATA_BLOCK

DATA_BLOCK "InstSimulationController"   // DB12
{ S7_Optimized_Access := 'TRUE' }
VERSION : 0.1
// stored: InstanceOfName Simulations-Controller
"Simulations-Controller"
BEGIN
END_DATA_BLOCK

// folder: 2. Machine

DATA_BLOCK "InstMachine"   // DB1000
{ S7_Optimized_Access := 'TRUE' }
VERSION : 0.1
// stored: InstanceOfName MachineControl
"MachineControl"
BEGIN
END_DATA_BLOCK

DATA_BLOCK "Machine"   // DB1001
{ S7_Optimized_Access := 'TRUE' }
VERSION : 0.1
   VAR
      safety : "typeMachineSafety";
      machine : "typeMachine";
      stations : "typeStations";
   END_VAR
BEGIN
   // stations.station[1] : FG01
   // stations.station[2] : FG02
   // stations.station[3] : FG03
   // stations.station[4] : FG04
   // stations.station[5] : FG05
   // stations.station[6] : Reserve
   // stations.station[7] : Reserve
   // stations.station[8] : Reserve
   // stations.station[9] : Reserve
   // stations.station[10] : Transport
   // stations.station[10].stepSeqs.stepSeq[1] : Stopper01
   // stations.station[10].stepSeqs.stepSeq[2] : Stopper02
   // stations.station[10].stepSeqs.stepSeq[3] : Lift01
   // stations.station[10].stepSeqs.stepSeq[4] : Stopper03
   // stations.station[10].stepSeqs.stepSeq[5] : Index01
   // stations.station[10].stepSeqs.stepSeq[6] : Index02
   // stations.station[10].stepSeqs.stepSeq[7] : Index03
   // stations.station[10].stepSeqs.stepSeq[8] : Index04
   // stations.station[10].stepSeqs.stepSeq[9] : Index05
   // stations.station[10].stepSeqs.stepSeq[10] : Stopper04
   // stations.station[10].stepSeqs.stepSeq[11] : Lift 2
END_DATA_BLOCK

DATA_BLOCK "ManualMovements"   // DB1005
{ S7_Optimized_Access := 'TRUE' }
VERSION : 0.1
BEGIN
END_DATA_BLOCK

// folder: 2. Machine/00_Alarms and Messages

DATA_BLOCK "Alarmserver"   // DB2
{ S7_Optimized_Access := 'TRUE' }
VERSION : 0.1
   VAR
      plc : Struct   // Meldungsspeicher für SPS
         machine : "typePlcErrMsg";
         fg_1 : "typePlcErrMsg";
         fg_2 : "typePlcErrMsg";
         fg_3 : "typePlcErrMsg";
         fg_4 : "typePlcErrMsg";
         fg_5 : "typePlcErrMsg";
         fg_transport : "typePlcErrMsg";
      END_STRUCT;
      hmi : Struct   // Meldungsspeicher für HMI
         machine : "typeHmiErrMsg";
         fg_1 : "typeHmiErrMsg";
         fg_2 : "typeHmiErrMsg";
         fg_3 : "typeHmiErrMsg";
         fg_4 : "typeHmiErrMsg";
         fg_5 : "typeHmiErrMsg";
         fg_transport : "typeHmiErrMsg";
      END_STRUCT;
   END_VAR
BEGIN
END_DATA_BLOCK

// folder: 2. Machine/01_FG01

DATA_BLOCK "InstFG01Control"   // DB1100
{ S7_Optimized_Access := 'TRUE' }
VERSION : 0.1
// stored: InstanceOfName FG01Control
"FG01Control"
BEGIN
END_DATA_BLOCK

DATA_BLOCK "FG01Parameter"   // DB1101
{ S7_Optimized_Access := 'TRUE' }
VERSION : 0.1
BEGIN
END_DATA_BLOCK

DATA_BLOCK "FG01Globals"   // DB1102
{ S7_Optimized_Access := 'TRUE' }
VERSION : 0.1
   VAR
      SQ1 : Struct
         readyForIndex : Bool;   // Freigabe für den Indexer zum Anheben
         isinHome : Bool;   // Grundstellung vorhanden
      END_STRUCT;
   END_VAR
BEGIN
END_DATA_BLOCK

DATA_BLOCK "FG01Actors"   // DB1103
{ S7_Optimized_Access := 'TRUE' }
VERSION : 0.1
   VAR
      Gripper : "typeActor_2Out2In";   // Greifer
      Plattform : "typeActor_2Out2In";   // Laserplattform
      ReaderWindow : "typeActor_2Out1In";   // Laserplattform
   END_VAR
BEGIN
END_DATA_BLOCK

// folder: 2. Machine/01_FG01/Stepsequences

DATA_BLOCK "InstSq_1.1"   // DB1111
{ S7_Optimized_Access := 'TRUE' }
VERSION : 0.1
// stored: InstanceOfName Sq_1.1
"Sq_1.1"
BEGIN
END_DATA_BLOCK

// folder: 2. Machine/02_FG02

DATA_BLOCK "InstFG02Control"   // DB1200
{ S7_Optimized_Access := 'TRUE' }
VERSION : 0.1
// stored: InstanceOfName FG02Control
"FG02Control"
BEGIN
END_DATA_BLOCK

DATA_BLOCK "FG02Globals"   // DB1202
{ S7_Optimized_Access := 'TRUE' }
VERSION : 0.1
   VAR
      SQ1 : Struct
         readyForIndex : Bool;   // Freigabe für den Indexer zum Anheben
         isInHome : Bool;   // Grundstellung vorhanden
      END_STRUCT;
   END_VAR
BEGIN
END_DATA_BLOCK

DATA_BLOCK "FG02Actors"   // DB1203
{ S7_Optimized_Access := 'TRUE' }
VERSION : 0.1
BEGIN
END_DATA_BLOCK

// folder: 2. Machine/02_FG02/Stepsequences

DATA_BLOCK "InstSq_2.1"   // DB1211
{ S7_Optimized_Access := 'TRUE' }
VERSION : 0.1
// stored: InstanceOfName Sq_2.1
"Sq_2.1"
BEGIN
END_DATA_BLOCK

// folder: 2. Machine/03_FG03

DATA_BLOCK "InstFG03Control"   // DB1300
{ S7_Optimized_Access := 'TRUE' }
VERSION : 0.1
// stored: InstanceOfName FG03Control
"FG03Control"
BEGIN
END_DATA_BLOCK

DATA_BLOCK "FG03Globals"   // DB1302
{ S7_Optimized_Access := 'TRUE' }
VERSION : 0.1
   VAR
      SQ1 : Struct
         readyForIndex : Bool;   // Freigabe für den Indexer zum Anheben
         isInHome : Bool;   // Grundstellung vorhanden
      END_STRUCT;
   END_VAR
BEGIN
END_DATA_BLOCK

DATA_BLOCK "FG03Actors"   // DB1303
{ S7_Optimized_Access := 'TRUE' }
VERSION : 0.1
   VAR
      AxisR1 : "typeActor_2Out2In";
      AxisX1 : "typeActor_2Out2In";
      AxisY1 : "typeActor_2Out2In";
      AxisX2 : "typeActor_2Out2In";
      AxisY2 : "typeActor_2Out2In";
      Gripper1 : "typeActor_2Out2In";
      Gripper2 : "typeActor_2Out2In";
   END_VAR
BEGIN
END_DATA_BLOCK

// folder: 2. Machine/03_FG03/Stepsequences

DATA_BLOCK "InstSq_3.1"   // DB1311
{ S7_Optimized_Access := 'TRUE' }
VERSION : 0.1
// stored: InstanceOfName Sq_3.1
"Sq_3.1"
BEGIN
END_DATA_BLOCK

// folder: 2. Machine/04_FG04

DATA_BLOCK "InstFG04Control"   // DB1400
{ S7_Optimized_Access := 'TRUE' }
VERSION : 0.1
// stored: InstanceOfName FG04Control
"FG04Control"
BEGIN
END_DATA_BLOCK

DATA_BLOCK "FG04Globals"   // DB1402
{ S7_Optimized_Access := 'TRUE' }
VERSION : 0.1
   VAR
      SQ1 : Struct
         readyForIndex : Bool;   // Freigabe für den Indexer zum Anheben
         isInHome : Bool;   // Grundstellung vorhanden
      END_STRUCT;
   END_VAR
BEGIN
END_DATA_BLOCK

DATA_BLOCK "FG04Actors"   // DB1403
{ S7_Optimized_Access := 'TRUE' }
VERSION : 0.1
   VAR
      AxisZ : "typeActor_2Out2In";
   END_VAR
BEGIN
END_DATA_BLOCK

// folder: 2. Machine/04_FG04/Stepsequences

DATA_BLOCK "InstSq_4.1"   // DB1411
{ S7_Optimized_Access := 'TRUE' }
VERSION : 0.1
// stored: InstanceOfName Sq_4.1
"Sq_4.1"
BEGIN
END_DATA_BLOCK

// folder: 2. Machine/05_FG05

DATA_BLOCK "InstFG05Control"   // DB1500
{ S7_Optimized_Access := 'TRUE' }
VERSION : 0.1
// stored: InstanceOfName FG05Control
"FG05Control"
BEGIN
END_DATA_BLOCK

DATA_BLOCK "FG05Globals"   // DB1502
{ S7_Optimized_Access := 'TRUE' }
VERSION : 0.1
   VAR
      SQ1 : Struct
         readyForIndex : Bool;   // Freigabe für den Indexer zum Anheben
         isInHome : Bool;   // Grundstellung vorhanden
      END_STRUCT;
   END_VAR
BEGIN
END_DATA_BLOCK

DATA_BLOCK "FG05Actors"   // DB1503
{ S7_Optimized_Access := 'TRUE' }
VERSION : 0.1
   VAR
      AxisR : "typeActor_2Out2In";
      AxisX : "typeActor_2Out2In";
      AxisZ1 : "typeActor_2Out2In";
      AxisZ2 : "typeActor_2Out2In";
      CapsSourceStopper : "typeActor_2Out1In";
      Gripper : "typeActor_2Out2In";
      Bunker : "typeActor_1Out0In";
      Conveyor : "typeActor_1Out0In";
   END_VAR
BEGIN
END_DATA_BLOCK

// folder: 2. Machine/05_FG05/Stepsequences

DATA_BLOCK "InstSq_5.1"   // DB1511
{ S7_Optimized_Access := 'TRUE' }
VERSION : 0.1
// stored: InstanceOfName Sq_5.1
"Sq_5.1"
BEGIN
END_DATA_BLOCK

// folder: 2. Machine/10_FG_Transport

DATA_BLOCK "InstTransportControl"   // DB2000
{ S7_Optimized_Access := 'TRUE' }
VERSION : 0.1
// stored: InstanceOfName TransportControl
"TransportControl"
BEGIN
END_DATA_BLOCK

DATA_BLOCK "TransportGlobals"   // DB2002
{ S7_Optimized_Access := 'TRUE' }
VERSION : 0.1
   VAR
      Index01 : Struct
         release : Bool;   // Startfreigabe für FG01 von Indexer
      END_STRUCT;
      Index02 : Struct
         release : Bool;   // Startfreigabe für FG02 von Indexer
      END_STRUCT;
      Index03 : Struct
         release : Bool;   // Startfreigabe für FG03 von Indexer
      END_STRUCT;
      Index04 : Struct
         release : Bool;   // Startfreigabe für FG04 von Indexer
      END_STRUCT;
      Index05 : Struct
         release : Bool;   // Startfreigabe für FG05 von Indexer
      END_STRUCT;
   END_VAR
BEGIN
END_DATA_BLOCK

DATA_BLOCK "TransportActors"   // DB2003
{ S7_Optimized_Access := 'TRUE' }
VERSION : 0.1
   VAR
      Gate_1 : "typeActor_1Out2In";
      Gate_2 : "typeActor_1Out2In";
      Index01_Lift : "typeActor_2Out2In";
      Index01_Stopper : "typeActor_1Out1In";
      Index02_Lift : "typeActor_2Out2In";
      Index02_Stopper : "typeActor_1Out1In";
      Index03_Lift : "typeActor_2Out2In";
      Index03_Stopper : "typeActor_1Out1In";
      Index04_Lift : "typeActor_2Out2In";
      Index04_Stopper : "typeActor_1Out1In";
      Index05_Lift : "typeActor_2Out2In";
      Index05_Stopper : "typeActor_1Out1In";
      Stopper01 : "typeActor_1Out1In";
      Stopper02 : "typeActor_1Out1In";
      Stopper03 : "typeActor_1Out1In";
      Stopper04 : "typeActor_1Out1In";
      Lift01_Lift : "typeActor_2Out2In";
      Lift01_Conv : "typeActor_2Out0In";
      Lift02_Lift : "typeActor_2Out2In";
      Lift02_Conv : "typeActor_2Out0In";
      Transport01_Conv : "typeActor_2Out0In";
      Transport02_Conv : "typeActor_2Out0In";
   END_VAR
BEGIN
END_DATA_BLOCK

// folder: 2. Machine/10_FG_Transport/Stepsequences

DATA_BLOCK "InstSq_Stopper01"   // DB2011
{ S7_Optimized_Access := 'TRUE' }
VERSION : 0.1
// stored: InstanceOfName Sq_Process_Stopper
"Sq_Process_Stopper"
BEGIN
END_DATA_BLOCK

DATA_BLOCK "InstSq_Stopper02"   // DB2012
{ S7_Optimized_Access := 'TRUE' }
VERSION : 0.1
// stored: InstanceOfName Sq_Process_Stopper
"Sq_Process_Stopper"
BEGIN
END_DATA_BLOCK

DATA_BLOCK "InstSq_Stopper03"   // DB2013
{ S7_Optimized_Access := 'TRUE' }
VERSION : 0.1
// stored: InstanceOfName Sq_Process_Stopper
"Sq_Process_Stopper"
BEGIN
END_DATA_BLOCK

DATA_BLOCK "InstSq_Stopper04"   // DB2014
{ S7_Optimized_Access := 'TRUE' }
VERSION : 0.1
// stored: InstanceOfName Sq_Process_Stopper
"Sq_Process_Stopper"
BEGIN
END_DATA_BLOCK

DATA_BLOCK "InstSq_Process_Lift1"   // DB2015
{ S7_Optimized_Access := 'TRUE' }
VERSION : 0.1
// stored: InstanceOfName Sq_Process_Lift
"Sq_Process_Lift"
BEGIN
END_DATA_BLOCK

DATA_BLOCK "InstSq_Process_Lift2"   // DB2016
{ S7_Optimized_Access := 'TRUE' }
VERSION : 0.1
// stored: InstanceOfName Sq_Process_Lift
"Sq_Process_Lift"
BEGIN
END_DATA_BLOCK

DATA_BLOCK "InstSq_Process_Index01"   // DB2017
{ S7_Optimized_Access := 'TRUE' }
VERSION : 0.1
// stored: InstanceOfName Sq_Process_IndexingUnit01
"Sq_Process_IndexingUnit01"
BEGIN
END_DATA_BLOCK

DATA_BLOCK "InstSq_Process_Index02"   // DB2018
{ S7_Optimized_Access := 'TRUE' }
VERSION : 0.1
// stored: InstanceOfName Sq_Process_IndexingUnit
"Sq_Process_IndexingUnit"
BEGIN
END_DATA_BLOCK

DATA_BLOCK "InstSq_Process_Index03"   // DB2019
{ S7_Optimized_Access := 'TRUE' }
VERSION : 0.1
// stored: InstanceOfName Sq_Process_IndexingUnit
"Sq_Process_IndexingUnit"
BEGIN
END_DATA_BLOCK

DATA_BLOCK "InstSq_Process_Index04"   // DB2020
{ S7_Optimized_Access := 'TRUE' }
VERSION : 0.1
// stored: InstanceOfName Sq_Process_IndexingUnit
"Sq_Process_IndexingUnit"
BEGIN
END_DATA_BLOCK

DATA_BLOCK "InstSq_Process_Index05"   // DB2021
{ S7_Optimized_Access := 'TRUE' }
VERSION : 0.1
// stored: InstanceOfName Sq_Process_IndexingUnit
"Sq_Process_IndexingUnit"
BEGIN
END_DATA_BLOCK

// folder: (top level)

ORGANIZATION_BLOCK "Main"   // OB1, LAD, ProgramCycle
TITLE = "Main Program Sweep (Cycle)"
{ S7_Optimized_Access := 'TRUE' }
VERSION : 0.1
   VAR_INPUT
      Initial_Call : Bool;   // Initial call of this OB
      Remanence : Bool;   // =True, if remanent data are available
   END_VAR
BEGIN

REGION Network 1: Inbetriebnahme-Merker
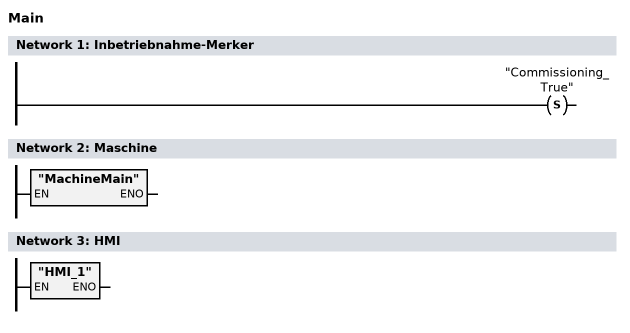
   RUNG wire#powerrail
      S_Coil( "Commissioning_True" )
   END_RUNG
   // the same network as SCL:
   "Commissioning_True" := TRUE;
END_REGION

REGION Network 2: Maschine
   RUNG wire#powerrail
      "MachineMain"()
   END_RUNG
   // the same network as SCL:
   "MachineMain"();
END_REGION

REGION Network 3: HMI
   RUNG wire#powerrail
      "HMI_1"()
   END_RUNG
   // the same network as SCL:
   "HMI_1"();
END_REGION
END_ORGANIZATION_BLOCK

// folder: 1. HMI

FUNCTION "HMI_1" : Void   // FC1001, FBD
TITLE = HMI
{ S7_Optimized_Access := 'TRUE' }
VERSION : 0.1
// Ersteller: Andreas Fast Automation
// E-Mail: automation@fast-andreas.de
// 
// Projekt dient zu Demonstrationszwecken und frei genutzt werden.
// 
// Bausteinbeschreibung:
BEGIN

REGION Network 1: Steuerung und Anzeige Einrichtbetrieb
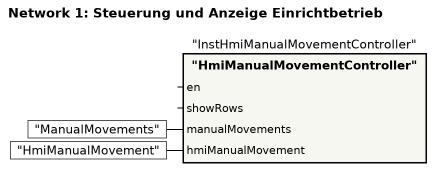
   "InstHmiManualMovementController"(manualMovements := "ManualMovements",   // "HmiManualMovementController"
                           hmiManualMovement := "HmiManualMovement");
END_REGION

REGION Network 2: Anzeige Schrittketteninformationen
END_REGION
END_FUNCTION

// folder: 10_Simulation (unused)

FUNCTION_BLOCK "Simulations-Controller"   // FB5, FBD
TITLE = Simulations-Controller (OEM abhängig)
{ S7_Optimized_Access := 'TRUE' }
VERSION : 0.1
   VAR_INPUT
      started : Bool;
   END_VAR
   VAR_OUTPUT
      synchronized : Bool;
      syncedStation10 : Bool;
      syncedStation20 : Bool;
   END_VAR
   VAR_IN_OUT
      iqudtSimInterface : "typeSimInterface";
   END_VAR
   VAR
      statStartedFlag : Bool;
      statResetSync : Bool;
   END_VAR
   VAR_TEMP
      tempDummy : Bool;
   END_VAR
   VAR_TEMP   // added for the SCL form of the ladder/FBD networks
      _w1 : Bool;
   END_VAR
BEGIN

REGION Network 1: Simulation wurde gestartet (SPS-Eingang)
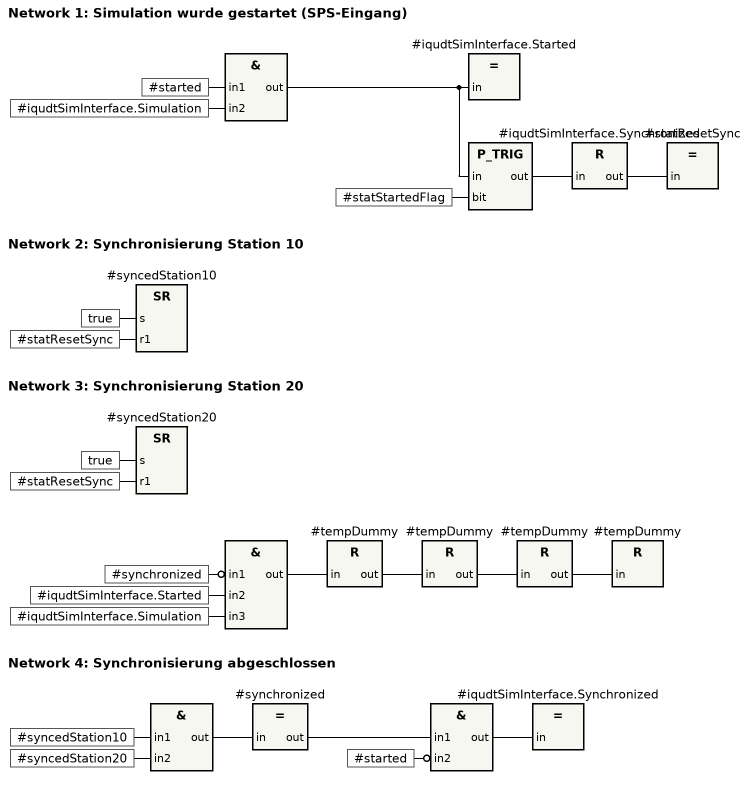
   #iqudtSimInterface.Started := #started AND #iqudtSimInterface.Simulation;
   #_w1 := #iqudtSimInterface.Started AND NOT #statStartedFlag;   // rising edge
   #statStartedFlag := #iqudtSimInterface.Started;
   IF #_w1 THEN #iqudtSimInterface.Synchronized := FALSE; END_IF;
   #statResetSync := #_w1;
END_REGION

REGION Network 2: Synchronisierung Station 10
   // Falls erforderlich, kann hier die Logik zur Synchronisierung der Station zwischen Simulation und SPS-Programm erfolgen.
   IF true THEN
       #syncedStation10 := TRUE;   // SR flip-flop
   END_IF;
   IF #statResetSync THEN #syncedStation10 := FALSE; END_IF;
END_REGION

REGION Network 3: Synchronisierung Station 20
   // Falls erforderlich, kann hier die Logik zur Synchronisierung der Station zwischen Simulation und SPS-Programm erfolgen.
   IF true THEN
       #syncedStation20 := TRUE;   // SR flip-flop
   END_IF;
   IF #statResetSync THEN #syncedStation20 := FALSE; END_IF;
   IF NOT #synchronized AND #iqudtSimInterface.Started AND #iqudtSimInterface.Simulation THEN
       #tempDummy := FALSE;
       #tempDummy := FALSE;
       #tempDummy := FALSE;
       #tempDummy := FALSE;
   END_IF;
END_REGION

REGION Network 4: Synchronisierung abgeschlossen
   #synchronized := #syncedStation10 AND #syncedStation20;
   #iqudtSimInterface.Synchronized := #synchronized AND NOT #started;
END_REGION
END_FUNCTION_BLOCK

FUNCTION "Simulation" : Void   // FC2, FBD
TITLE = Simulation
{ S7_Optimized_Access := 'TRUE' }
VERSION : 0.1
BEGIN

REGION Network 1: Simulation
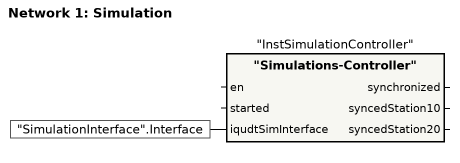
   "InstSimulationController"(iqudtSimInterface := "SimulationInterface".Interface);   // "Simulations-Controller"
END_REGION
END_FUNCTION

// folder: 2. Machine

FUNCTION "MachineMain" : Void   // FC1000, FBD
TITLE = Machine
{ S7_Optimized_Access := 'TRUE' }
VERSION : 0.1
// Ersteller: Andreas Fast Automation
// E-Mail: automation@fast-andreas.de
// 
// Projekt dient zu Demonstrationszwecken und frei genutzt werden.
BEGIN

REGION Network 1: Machine
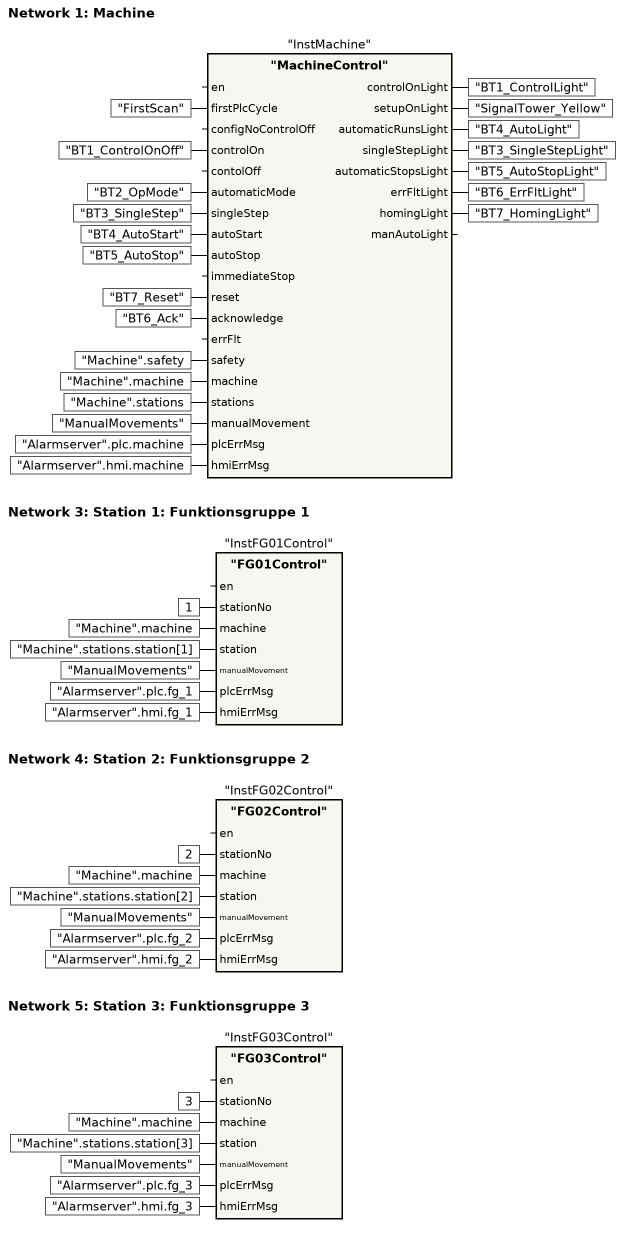
   "InstMachine"(firstPlcCycle := "FirstScan",   // "MachineControl"
                 controlOn := "BT1_ControlOnOff",
                 automaticMode := "BT2_OpMode",
                 singleStep := "BT3_SingleStep",
                 autoStart := "BT4_AutoStart",
                 autoStop := "BT5_AutoStop",
                 reset := "BT7_Reset",
                 acknowledge := "BT6_Ack",
                 safety := "Machine".safety,
                 machine := "Machine".machine,
                 stations := "Machine".stations,
                 manualMovement := "ManualMovements",
                 plcErrMsg := "Alarmserver".plc.machine,
                 hmiErrMsg := "Alarmserver".hmi.machine,
                 controlOnLight => "BT1_ControlLight",
                 setupOnLight => "SignalTower_Yellow",
                 automaticRunsLight => "BT4_AutoLight",
                 singleStepLight => "BT3_SingleStepLight",
                 automaticStopsLight => "BT5_AutoStopLight",
                 errFltLight => "BT6_ErrFltLight",
                 homingLight => "BT7_HomingLight");
END_REGION

REGION Network 2: Ampel
END_REGION

REGION Network 3: Station 1: Funktionsgruppe 1
   "InstFG01Control"(stationNo := 1,   // "FG01Control"
                     machine := "Machine".machine,
                     station := "Machine".stations.station[1],
                     manualMovement := "ManualMovements",
                     plcErrMsg := "Alarmserver".plc.fg_1,
                     hmiErrMsg := "Alarmserver".hmi.fg_1);
END_REGION

REGION Network 4: Station 2: Funktionsgruppe 2
   "InstFG02Control"(stationNo := 2,   // "FG02Control"
                     machine := "Machine".machine,
                     station := "Machine".stations.station[2],
                     manualMovement := "ManualMovements",
                     plcErrMsg := "Alarmserver".plc.fg_2,
                     hmiErrMsg := "Alarmserver".hmi.fg_2);
END_REGION

REGION Network 5: Station 3: Funktionsgruppe 3
   "InstFG03Control"(stationNo := 3,   // "FG03Control"
                     machine := "Machine".machine,
                     station := "Machine".stations.station[3],
                     manualMovement := "ManualMovements",
                     plcErrMsg := "Alarmserver".plc.fg_3,
                     hmiErrMsg := "Alarmserver".hmi.fg_3);
END_REGION

REGION Network 6: Station 4: Funktionsgruppe 4
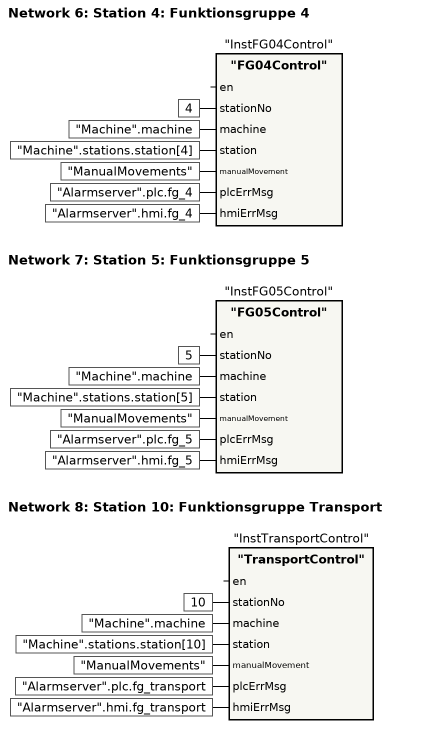
   "InstFG04Control"(stationNo := 4,   // "FG04Control"
                     machine := "Machine".machine,
                     station := "Machine".stations.station[4],
                     manualMovement := "ManualMovements",
                     plcErrMsg := "Alarmserver".plc.fg_4,
                     hmiErrMsg := "Alarmserver".hmi.fg_4);
END_REGION

REGION Network 7: Station 5: Funktionsgruppe 5
   "InstFG05Control"(stationNo := 5,   // "FG05Control"
                     machine := "Machine".machine,
                     station := "Machine".stations.station[5],
                     manualMovement := "ManualMovements",
                     plcErrMsg := "Alarmserver".plc.fg_5,
                     hmiErrMsg := "Alarmserver".hmi.fg_5);
END_REGION

REGION Network 8: Station 10: Funktionsgruppe Transport
   "InstTransportControl"(stationNo := 10,   // "TransportControl"
                          machine := "Machine".machine,
                          station := "Machine".stations.station[10],
                          manualMovement := "ManualMovements",
                          plcErrMsg := "Alarmserver".plc.fg_transport,
                          hmiErrMsg := "Alarmserver".hmi.fg_transport);
END_REGION
END_FUNCTION

// folder: 2. Machine/00_Alarms and Messages

FUNCTION "MachineAlarms" : Void   // FC1009, LAD
TITLE = Störmeldungen Maschine
{ S7_Optimized_Access := 'TRUE' }
VERSION : 0.1
// Ersteller: Andreas Fast Automation
// E-Mail: automation@fast-andreas.de
// 
// Projekt dient zu Demonstrationszwecken und frei genutzt werden.
// 
// Bausteinbeschreibung: 
// Störmeldungen werden über die Quittierung zurückgesetzt.
   VAR_IN_OUT
      machine : "typeMachine";
      alarms : "typePlcErrors";
   END_VAR
BEGIN

REGION Network 1: Initialisierung für die Einrichtbewegungen ist fehlerhaft
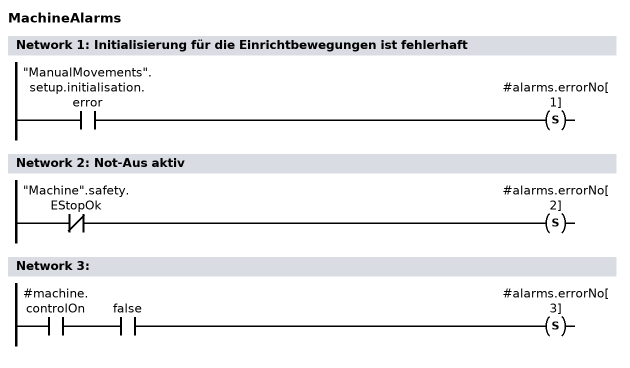
   RUNG wire#powerrail
      Contact( "ManualMovements".setup.initialisation.error )
      S_Coil( #alarms.errorNo[1] )
   END_RUNG
   // the same network as SCL:
   IF "ManualMovements".setup.initialisation.error THEN #alarms.errorNo[1] := TRUE; END_IF;
END_REGION

REGION Network 2: Not-Aus aktiv
   RUNG wire#powerrail
      I_Contact( "Machine".safety.EStopOk )
      S_Coil( #alarms.errorNo[2] )
   END_RUNG
   // the same network as SCL:
   IF NOT "Machine".safety.EStopOk THEN #alarms.errorNo[2] := TRUE; END_IF;
END_REGION

REGION Network 3
   RUNG wire#powerrail
      Contact( #machine.controlOn )
      Contact( false )
      S_Coil( #alarms.errorNo[3] )
   END_RUNG
   // the same network as SCL:
   IF #machine.controlOn AND false THEN #alarms.errorNo[3] := TRUE; END_IF;
END_REGION
END_FUNCTION

FUNCTION "MachineMessages" : Void   // FC1010, LAD
TITLE = Meldungen Maschine
{ S7_Optimized_Access := 'TRUE' }
VERSION : 0.1
// Ersteller: Andreas Fast Automation
// E-Mail: automation@fast-andreas.de
// 
// Projekt dient zu Demonstrationszwecken und frei genutzt werden.
// 
// Bausteinbeschreibung: 
// Störmeldungen werden über die Quittierung zurückgesetzt.
   VAR_IN_OUT
      machine : "typeMachine";
      messages : "typePlcMessages";
   END_VAR
BEGIN

REGION Network 1: Maschine ist ausgeschaltet
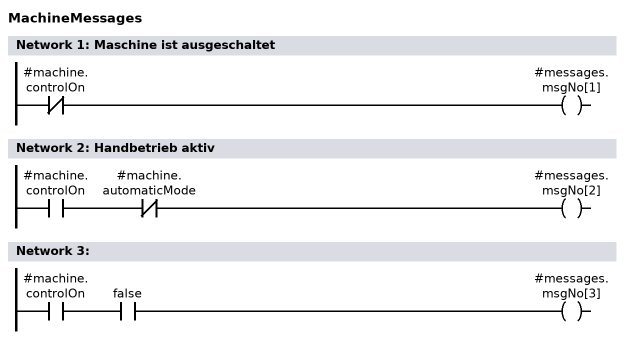
   RUNG wire#powerrail
      I_Contact( #machine.controlOn )
      Coil( #messages.msgNo[1] )
   END_RUNG
   // the same network as SCL:
   #messages.msgNo[1] := NOT #machine.controlOn;
END_REGION

REGION Network 2: Handbetrieb aktiv
   RUNG wire#powerrail
      Contact( #machine.controlOn )
      I_Contact( #machine.automaticMode )
      Coil( #messages.msgNo[2] )
   END_RUNG
   // the same network as SCL:
   #messages.msgNo[2] := #machine.controlOn AND NOT #machine.automaticMode;
END_REGION

REGION Network 3
   RUNG wire#powerrail
      Contact( #machine.controlOn )
      Contact( false )
      Coil( #messages.msgNo[3] )
   END_RUNG
   // the same network as SCL:
   #messages.msgNo[3] := #machine.controlOn AND false;
END_REGION
END_FUNCTION

// folder: 2. Machine/01_FG01

FUNCTION_BLOCK "FG01Control"   // FB1100, FBD
TITLE = Station 1 Hauptaufruf
{ S7_Optimized_Access := 'TRUE' }
VERSION : 0.1
// Ersteller: Andreas Fast Automation
// E-Mail: automation@fast-andreas.de
// 
// Projekt dient zu Demonstrationszwecken und frei genutzt werden.
// 
// Bausteinbeschreibung:
   VAR_INPUT
      stationNo : Int := 1;   // Stationsnummer
   END_VAR
   VAR_IN_OUT
      machine : "typeMachine";
      station : "typeStation";
      manualMovement : "typeManualMovements";
      plcErrMsg : "typePlcErrMsg";
      hmiErrMsg : "typeHmiErrMsg";
   END_VAR
   VAR
      instStationControl : "StationControl";
      instActorControl : "FG01ActorControl";
   END_VAR
   VAR_TEMP
      tempSafetyOk : Bool;
   END_VAR
BEGIN

REGION Network 1: Stationssteuerung
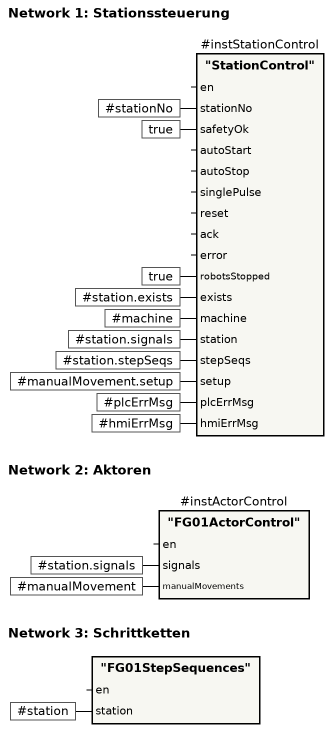
   #instStationControl(stationNo := #stationNo,   // "StationControl"
                       safetyOk := true,
                       robotsStopped := true,
                       exists := #station.exists,
                       machine := #machine,
                       station := #station.signals,
                       stepSeqs := #station.stepSeqs,
                       setup := #manualMovement.setup,
                       plcErrMsg := #plcErrMsg,
                       hmiErrMsg := #hmiErrMsg);
END_REGION

REGION Network 2: Aktoren
   #instActorControl(signals := #station.signals, manualMovements := #manualMovement);   // "FG01ActorControl"
END_REGION

REGION Network 3: Schrittketten
   "FG01StepSequences"(station := #station);
END_REGION
END_FUNCTION_BLOCK

FUNCTION_BLOCK "FG01ActorControl"   // FB1102, FBD
TITLE = Aktoransteuerung
{ S7_Optimized_Access := 'TRUE' }
VERSION : 0.1
// Ersteller: Andreas Fast Automation
// E-Mail: automation@fast-andreas.de
// 
// Projekt dient zu Demonstrationszwecken und frei genutzt werden.
// 
// Bausteinbeschreibung:
   VAR_IN_OUT
      signals : "typeStationSignals";
      manualMovements : "typeManualMovements";
   END_VAR
   VAR
      sinstGripper : "Cylinder_2Out2In";
      sinstPlattform : "Cylinder_2Out2In";
      sinstReaderWindow : "Cylinder_2Out1In (ungetestet)";
      instActorReserved4 : "Actor_Reserved";
      instActorReserved5 : "Actor_Reserved";
      instActorReserved6 : "Actor_Reserved";
      instActorReserved7 : "Actor_Reserved";
      instActorReserved8 : "Actor_Reserved";
   END_VAR
BEGIN

REGION Network 1: Gripper
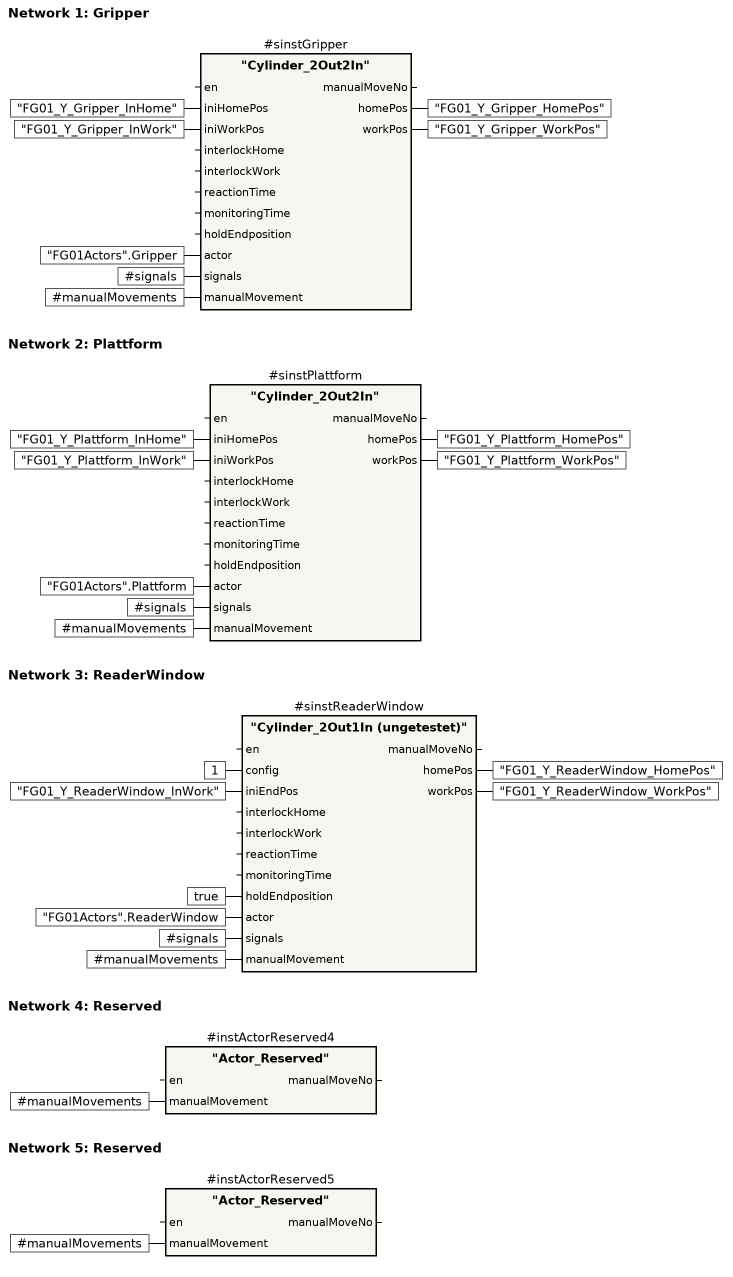
   #sinstGripper(iniHomePos := "FG01_Y_Gripper_InHome",   // "Cylinder_2Out2In"
                 iniWorkPos := "FG01_Y_Gripper_InWork",
                 actor := "FG01Actors".Gripper,
                 signals := #signals,
                 manualMovement := #manualMovements,
                 homePos => "FG01_Y_Gripper_HomePos",
                 workPos => "FG01_Y_Gripper_WorkPos");
END_REGION

REGION Network 2: Plattform
   #sinstPlattform(iniHomePos := "FG01_Y_Plattform_InHome",   // "Cylinder_2Out2In"
                   iniWorkPos := "FG01_Y_Plattform_InWork",
                   actor := "FG01Actors".Plattform,
                   signals := #signals,
                   manualMovement := #manualMovements,
                   homePos => "FG01_Y_Plattform_HomePos",
                   workPos => "FG01_Y_Plattform_WorkPos");
END_REGION

REGION Network 3: ReaderWindow
   #sinstReaderWindow(config := 1,   // "Cylinder_2Out1In (ungetestet)"
                      iniEndPos := "FG01_Y_ReaderWindow_InWork",
                      holdEndposition := true,
                      actor := "FG01Actors".ReaderWindow,
                      signals := #signals,
                      manualMovement := #manualMovements,
                      homePos => "FG01_Y_ReaderWindow_HomePos",
                      workPos => "FG01_Y_ReaderWindow_WorkPos");
END_REGION

REGION Network 4: Reserved
   #instActorReserved4(manualMovement := #manualMovements);   // "Actor_Reserved"
END_REGION

REGION Network 5: Reserved
   #instActorReserved5(manualMovement := #manualMovements);   // "Actor_Reserved"
END_REGION

REGION Network 6: Reserved
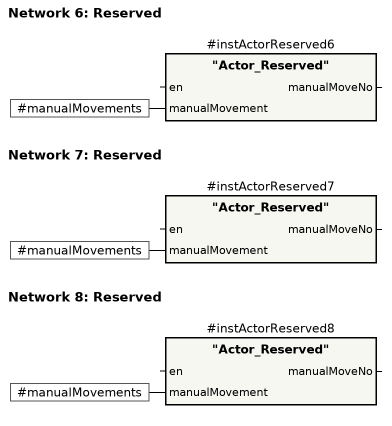
   #instActorReserved6(manualMovement := #manualMovements);   // "Actor_Reserved"
END_REGION

REGION Network 7: Reserved
   #instActorReserved7(manualMovement := #manualMovements);   // "Actor_Reserved"
END_REGION

REGION Network 8: Reserved
   #instActorReserved8(manualMovement := #manualMovements);   // "Actor_Reserved"
END_REGION
END_FUNCTION_BLOCK

// folder: 2. Machine/01_FG01/Stepsequences

FUNCTION_BLOCK "Sq_1.1"   // FB1111, GRAPH_PLUS
{ S7_Optimized_Access := 'TRUE' }
VERSION : 0.1
   VAR_INPUT
      OFF_SQ : Bool := false;   // Kette ausschalten
      INIT_SQ : Bool := false;   // Kette in Initialzustand versetzen
      ACK_EF : Bool := false;   // Alle Fehler und Störungen quittieren
      S_PREV : Bool := false;   // Vorherigen Schritt am Parameter S_NO ausgeben
      S_NEXT : Bool := false;   // Nächsten Schritt am Parameter S_NO anzeigen
      SW_AUTO : Bool := false;   // Automatischer Betrieb
      SW_TAP : Bool := false;   // Halbautomatisch/Weiterschalten mit Transition
      SW_TOP : Bool := false;   // Halbautomatisch/Ignoriere Transition
      SW_MAN : Bool := false;   // Handbetrieb
      S_SEL : Int := 0;   // Schritt auswählen, der an S_NO ausgegeben werden soll
      S_ON : Bool := false;   // Schritt aktivieren, der an Parameter S_NO anliegt
      S_OFF : Bool := false;   // Schritt deaktivieren, der an Parameter S_NO anliegt
      T_PUSH : Bool := false;   // Schaltfreigabe für Transition im halbautomatischen Betrieb
      itMaxRuntime : Time := t#10s;   // Maximale Laufzeit für diesen Prozess
   END_VAR
   VAR_OUTPUT
      S_NO : Int := 0;   // Schrittnummer
      S_MORE : Bool := false;   // Weitere Schritte sind vorhanden und können in S_NO angezeigt werden.
      S_ACTIVE : Bool := false;   // Schritt, der an Parameter S_NO angezeigt wird, ist aktiv
      ERR_FLT : Bool := false;   // Sammelfehler Interlock oder Supervision
      AUTO_ON : Bool := false;   // Automatischer Betrieb eingeschaltet
      TAP_ON : Bool := false;   // Halbautomatischer Betrieb/Schritt mit Transition eingeschaltet
      TOP_ON : Bool := false;   // Halbautomatischer Betrieb/Ignoriere Transition eingeschaltet
      MAN_ON : Bool := false;   // Handbetrieb eingeschaltet
      qxIsActive : Bool;   // Schrittkette läuft
      qxIsInHome : Bool;   // steht in Grundstellung
   END_VAR
   VAR_IN_OUT
      signals : "typeStationSignals";   // Stationssteuersignale
      sq : "typeStepSequence";   // Schrittkettensteuersignale
   END_VAR
   VAR
      sstReleaseCycle : Struct
         ErrorAck : Bool;
         No_LastCycle : Int;
         T : Time;   // Aktive Zeit des ReleaseCycle
         Tck : Time;
         TckPrev : Time;
      END_STRUCT;
      HMI_INFO : Array[0..8] of UInt;
      IF_PAR : G7_IfParPlus_V6;
      RT_DATA : G7_RTDataPlus_V6;   // Interner Datenbereich
      Automatikablauf : G7_TransitionPlus_V6;   // Transitionsstruktur
      Freigabe : G7_TransitionPlus_V6;   // Transitionsstruktur
      Trans3 : G7_TransitionPlus_V6;   // Transitionsstruktur
      Fertig : G7_TransitionPlus_V6;   // Transitionsstruktur
      Grundstellungsfahrt : G7_TransitionPlus_V6;   // Transitionsstruktur
      GST_Aktiv : G7_TransitionPlus_V6;   // Transitionsstruktur
      GST_Beendet : G7_TransitionPlus_V6;   // Transitionsstruktur
      Beendet : G7_TransitionPlus_V6;   // Transitionsstruktur
      DoneToIndexer : G7_TransitionPlus_V6;   // Transitionsstruktur / Transition structure
      GS_GripperInHome : G7_TransitionPlus_V6;   // Transitionsstruktur / Transition structure
      GS_PlattformInHome : G7_TransitionPlus_V6;   // Transitionsstruktur / Transition structure
      GS_ReaderWindowInHome : G7_TransitionPlus_V6;   // Transitionsstruktur / Transition structure
      PlattformIsInWork : G7_TransitionPlus_V6;   // Transitionsstruktur / Transition structure
      ReaderWindowInWork : G7_TransitionPlus_V6;   // Transitionsstruktur / Transition structure
      GripperInWork : G7_TransitionPlus_V6;   // Transitionsstruktur / Transition structure
      GripperInHome : G7_TransitionPlus_V6;   // Transitionsstruktur / Transition structure
      PlattformIsInWork_1 : G7_TransitionPlus_V6;   // Transitionsstruktur / Transition structure
      ReaderWindowInHome : G7_TransitionPlus_V6;   // Transitionsstruktur / Transition structure
      JogT1 : G7_TransitionPlus_V6;   // Transitionsstruktur / Transition structure
      JogT2 : G7_TransitionPlus_V6;   // Transitionsstruktur / Transition structure
      JogT3 : G7_TransitionPlus_V6;   // Transitionsstruktur / Transition structure
      JogT4 : G7_TransitionPlus_V6;   // Transitionsstruktur / Transition structure
      Trans34 : G7_TransitionPlus_V6;   // Transitionsstruktur / Transition structure
      JogT5 : G7_TransitionPlus_V6;   // Transitionsstruktur / Transition structure
      Initialschritt : G7_StepPlus_V6;   // Schrittstruktur
      Grundstellung : G7_StepPlus_V6;   // Schrittstruktur
      SK_läuft : G7_StepPlus_V6;   // Schrittstruktur
      Fertigmeldung : G7_StepPlus_V6;   // Schrittstruktur
      "Start Grundstellungsfahrt" : G7_StepPlus_V6;   // Schrittstruktur
      "Fertig Grundstellungsfahrt" : G7_StepPlus_V6;   // Schrittstruktur
      Ende : G7_StepPlus_V6;   // Schrittstruktur
      ResetRelease : G7_StepPlus_V6;   // Schrittstruktur / Step structure
      GS_GripperHome : G7_StepPlus_V6;   // Schrittstruktur / Step structure
      GS_PlattformHome : G7_StepPlus_V6;   // Schrittstruktur / Step structure
      GS_ReaderWindowHome : G7_StepPlus_V6;   // Schrittstruktur / Step structure
      PlattformToWork : G7_StepPlus_V6;   // Schrittstruktur / Step structure
      ReaderWindowToWork : G7_StepPlus_V6;   // Schrittstruktur / Step structure
      GripperToWork : G7_StepPlus_V6;   // Schrittstruktur / Step structure
      GripperToHome : G7_StepPlus_V6;   // Schrittstruktur / Step structure
      PlattformToHome : G7_StepPlus_V6;   // Schrittstruktur / Step structure
      ReaderWindowToHome : G7_StepPlus_V6;   // Schrittstruktur / Step structure
      JogS1 : G7_StepPlus_V6;   // Schrittstruktur / Step structure
      JogS2 : G7_StepPlus_V6;   // Schrittstruktur / Step structure
      JogS3 : G7_StepPlus_V6;   // Schrittstruktur / Step structure
      JogS4 : G7_StepPlus_V6;   // Schrittstruktur / Step structure
      Cam : G7_StepPlus_V6;   // Schrittstruktur / Step structure
      JogS5 : G7_StepPlus_V6;   // Schrittstruktur / Step structure
      SINI : Array[0..1] of USInt;
      LSTT : Array[0..23] of USInt;
      ATAJ : Array[0..23] of USInt;
      ATAB : Array[0..23] of USInt;
      PSTT : Array[0..23] of USInt;
      NSTT : Array[0..23] of USInt;
      ASSJ : Array[0..22] of USInt;
      ASSB : Array[0..22] of USInt;
      PTTS : Array[0..22] of USInt;
      NTTS : Array[0..22] of USInt;
      SW_SQTS : Array[0..22] of USInt;
      SWITCH : Array[0..1] of USInt;
      TVX : Array[0..3] of USInt;
      TTX : Array[0..3] of USInt;
      TSX : Array[0..1] of USInt;
      S00X : Array[0..1] of USInt;
      SOFFX : Array[0..1] of USInt;
      SONX : Array[0..1] of USInt;
      SAX : Array[0..1] of USInt;
      SERRX : Array[0..23] of USInt;
      SMX : Array[0..23] of USInt;
      S0X : Array[0..23] of USInt;
      S1X : Array[0..23] of USInt;
      IL_ALARM_INST : Diag_Alarm;
      SUP_ALARM_INST : Diag_Alarm;
      STEP_TIME_ALARM_INST : Diag_Alarm;
      IEC_TIMER_INST : IEC_TIMER;
      TRANSACTION_FLAG : Bool := false;
   END_VAR
   VAR_TEMP
      txStartCondition : Bool;
      tdTckDiff : DInt;
   END_VAR
   VAR_TEMP   // added for the SCL form of the ladder/FBD networks
      _w1 : Bool;
      _w2 : Bool;
   END_VAR
   // SINI[0] := 2;
   // LSTT[0] := 255;
   // LSTT[1] := 255;
   // LSTT[2] := 255;
   // LSTT[3] := 255;
   // LSTT[4] := 255;
   // LSTT[5] := 255;
   // LSTT[6] := 255;
   // LSTT[7] := 1;
   // ATAJ[1] := 1;
   // ATAJ[2] := 2;
   // ATAJ[3] := 6;
   // ATAJ[4] := 4;
   // ATAJ[5] := 5;
   // ATAJ[6] := 3;
   // ATAJ[7] := 7;
   // ATAB[0] := 4;
   // ATAB[1] := 1;
   // ATAB[2] := 2;
   // ATAB[3] := 3;
   // ATAB[5] := 5;
   // ATAB[6] := 6;
   // ATAB[7] := 7;
   // PSTT[1] := 1;
   // PSTT[2] := 2;
   // PSTT[3] := 3;
   // PSTT[5] := 4;
   // PSTT[6] := 5;
   // PSTT[7] := 6;
   // NSTT[0] := 1;
   // NSTT[1] := 2;
   // NSTT[2] := 13;
   // NSTT[3] := 6;
   // NSTT[4] := 4;
   // NSTT[5] := 8;
   // NSTT[6] := 6;
   // NSTT[7] := 1;
   // ASSJ[1] := 1;
   // ASSJ[2] := 2;
   // ASSJ[3] := 3;
   // ASSJ[4] := 4;
   // ASSJ[5] := 5;
   // ASSJ[6] := 6;
   // ASSB[1] := 1;
   // ASSB[2] := 2;
   // ASSB[3] := 3;
   // ASSB[4] := 4;
   // ASSB[5] := 5;
   // ASSB[6] := 6;
   // PTTS[0] := 255;
   // PTTS[2] := 1;
   // PTTS[3] := 8;
   // PTTS[4] := 4;
   // PTTS[5] := 11;
   // PTTS[6] := 3;
   // NTTS[1] := 1;
   // NTTS[2] := 2;
   // NTTS[3] := 3;
   // NTTS[4] := 5;
   // NTTS[5] := 6;
   // NTTS[6] := 7;
   // SW_SQTS[1] := 1;
   // SW_SQTS[2] := 1;
   // SW_SQTS[3] := 1;
   // SW_SQTS[4] := 2;
   // SW_SQTS[5] := 2;
   // SW_SQTS[6] := 3;
   // TVX[0] := 16#1;
   // TTX[0] := 16#1;
   // TSX[0] := 16#1;
   // S00X[0] := 16#1;
   // SOFFX[0] := 16#1;
   // SONX[0] := 16#1;
   // SAX[0] := 16#1;
   // SERRX[0] := 16#1;
   // SMX[0] := 16#1;
   // S0X[0] := 16#1;
   // S1X[0] := 16#1;
   // LSTT[8] := 255;
   // ATAJ[8] := 8;
   // ATAB[8] := 8;
   // PSTT[8] := 7;
   // NSTT[8] := 3;
   // ASSJ[7] := 7;
   // ASSB[7] := 7;
   // PTTS[7] := 17;
   // NTTS[7] := 8;
   // SW_SQTS[7] := 1;
   // LSTT[9] := 255;
   // LSTT[10] := 255;
   // LSTT[11] := 255;
   // ATAJ[9] := 9;
   // ATAJ[10] := 10;
   // ATAJ[11] := 11;
   // ATAB[9] := 9;
   // ATAB[10] := 10;
   // ATAB[11] := 11;
   // PSTT[9] := 8;
   // PSTT[10] := 9;
   // PSTT[11] := 10;
   // NSTT[9] := 9;
   // NSTT[10] := 10;
   // NSTT[11] := 5;
   // ASSJ[8] := 8;
   // ASSJ[9] := 9;
   // ASSJ[10] := 10;
   // ASSB[8] := 8;
   // ASSB[9] := 9;
   // ASSB[10] := 10;
   // PTTS[8] := 5;
   // PTTS[9] := 9;
   // PTTS[10] := 10;
   // NTTS[8] := 9;
   // NTTS[9] := 10;
   // NTTS[10] := 11;
   // SW_SQTS[8] := 2;
   // SW_SQTS[9] := 2;
   // SW_SQTS[10] := 2;
   // LSTT[12] := 255;
   // LSTT[13] := 255;
   // LSTT[14] := 255;
   // LSTT[15] := 255;
   // ATAJ[12] := 12;
   // ATAJ[13] := 13;
   // ATAJ[14] := 14;
   // ATAJ[15] := 15;
   // ATAB[12] := 12;
   // ATAB[13] := 13;
   // ATAB[14] := 14;
   // ATAB[15] := 15;
   // PSTT[12] := 11;
   // PSTT[13] := 12;
   // PSTT[14] := 13;
   // PSTT[15] := 14;
   // NSTT[12] := 18;
   // NSTT[13] := 19;
   // NSTT[14] := 17;
   // NSTT[15] := 16;
   // ASSJ[11] := 11;
   // ASSJ[12] := 12;
   // ASSJ[13] := 13;
   // ASSJ[14] := 14;
   // ASSB[11] := 11;
   // ASSB[12] := 12;
   // ASSB[13] := 13;
   // ASSB[14] := 14;
   // PTTS[11] := 18;
   // PTTS[12] := 19;
   // PTTS[13] := 2;
   // PTTS[14] := 23;
   // NTTS[11] := 12;
   // NTTS[12] := 13;
   // NTTS[13] := 14;
   // NTTS[14] := 15;
   // SW_SQTS[11] := 1;
   // SW_SQTS[12] := 1;
   // SW_SQTS[13] := 1;
   // SW_SQTS[14] := 1;
   // LSTT[16] := 255;
   // ATAJ[16] := 16;
   // ATAB[16] := 16;
   // PSTT[16] := 15;
   // NSTT[16] := 22;
   // ASSJ[15] := 15;
   // ASSB[15] := 15;
   // PTTS[15] := 21;
   // NTTS[15] := 16;
   // SW_SQTS[15] := 1;
   // LSTT[17] := 255;
   // LSTT[18] := 255;
   // LSTT[19] := 255;
   // LSTT[20] := 255;
   // LSTT[21] := 255;
   // LSTT[22] := 255;
   // ATAJ[17] := 17;
   // ATAJ[18] := 18;
   // ATAJ[19] := 19;
   // ATAJ[20] := 20;
   // ATAJ[21] := 21;
   // ATAJ[22] := 22;
   // ATAB[17] := 17;
   // ATAB[18] := 18;
   // ATAB[19] := 19;
   // ATAB[20] := 20;
   // ATAB[21] := 21;
   // ATAB[22] := 22;
   // PSTT[17] := 16;
   // PSTT[18] := 17;
   // PSTT[19] := 18;
   // PSTT[20] := 19;
   // PSTT[21] := 20;
   // PSTT[22] := 21;
   // NSTT[17] := 7;
   // NSTT[18] := 11;
   // NSTT[19] := 12;
   // NSTT[20] := 21;
   // NSTT[21] := 15;
   // NSTT[22] := 20;
   // ASSJ[16] := 16;
   // ASSJ[17] := 17;
   // ASSJ[18] := 18;
   // ASSJ[19] := 19;
   // ASSJ[20] := 20;
   // ASSJ[21] := 21;
   // ASSB[16] := 16;
   // ASSB[17] := 17;
   // ASSB[18] := 18;
   // ASSB[19] := 19;
   // ASSB[20] := 20;
   // ASSB[21] := 21;
   // PTTS[16] := 15;
   // PTTS[17] := 14;
   // PTTS[18] := 12;
   // PTTS[19] := 13;
   // PTTS[20] := 22;
   // PTTS[21] := 20;
   // NTTS[16] := 17;
   // NTTS[17] := 18;
   // NTTS[18] := 19;
   // NTTS[19] := 20;
   // NTTS[20] := 21;
   // NTTS[21] := 22;
   // SW_SQTS[16] := 1;
   // SW_SQTS[17] := 1;
   // SW_SQTS[18] := 1;
   // SW_SQTS[19] := 1;
   // SW_SQTS[20] := 1;
   // SW_SQTS[21] := 1;
   // LSTT[23] := 255;
   // ATAJ[23] := 23;
   // ATAB[23] := 23;
   // PSTT[23] := 22;
   // NSTT[23] := 14;
   // ASSJ[22] := 22;
   // ASSB[22] := 22;
   // PTTS[22] := 16;
   // NTTS[22] := 23;
   // SW_SQTS[22] := 1;
BEGIN
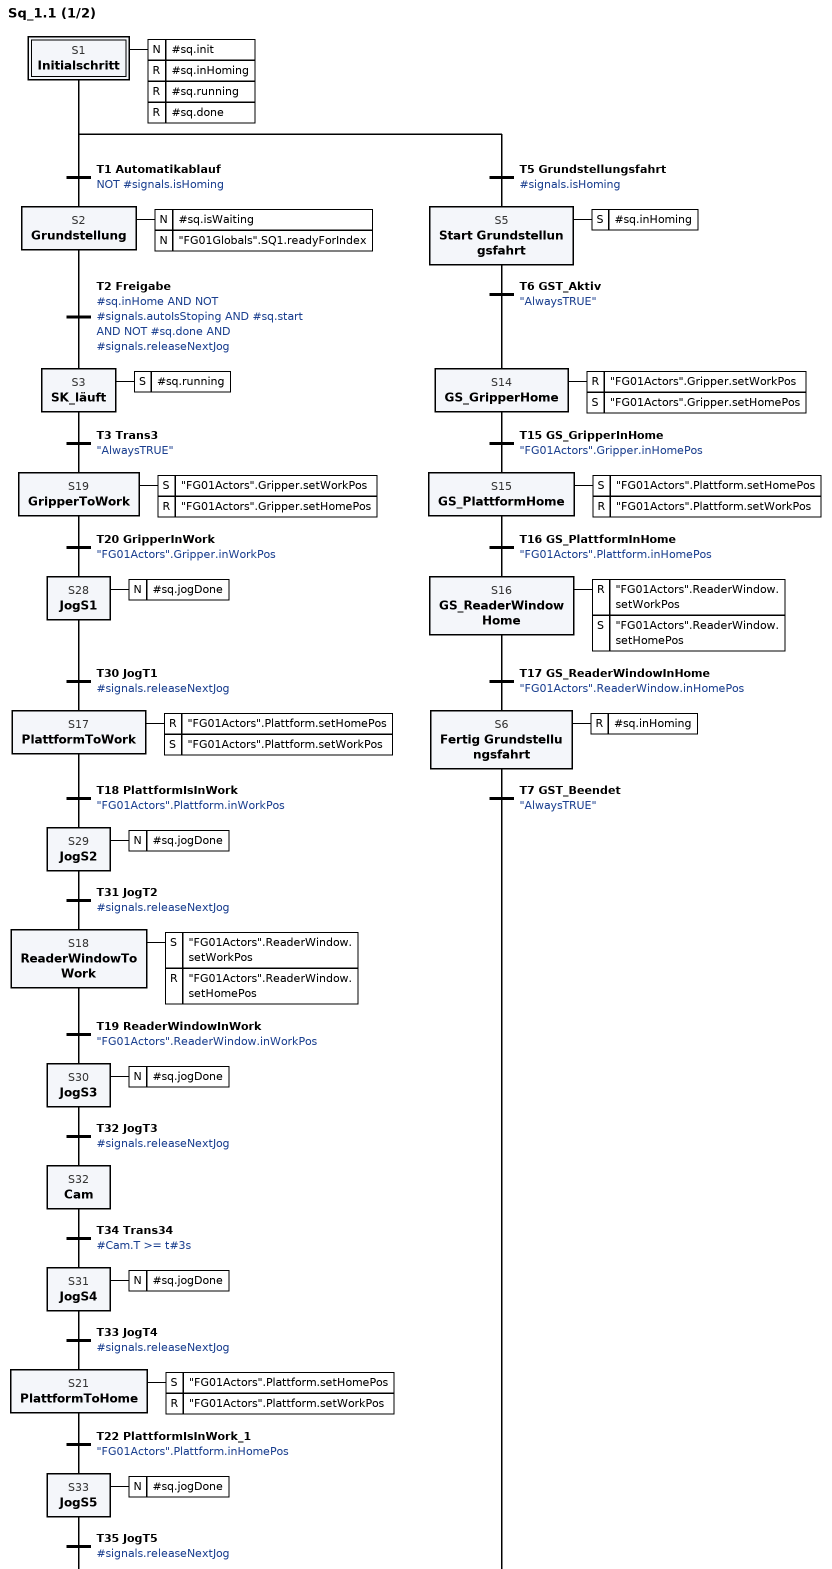
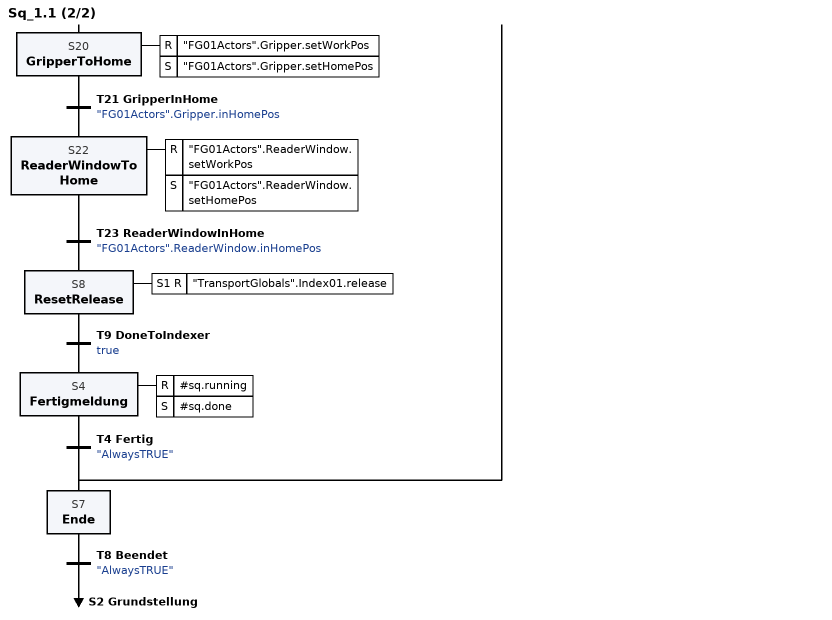
   // permanent pre-instructions
   NETWORK 1
   TITLE = Schrittkette verfügbar
      #sq.exists := true;
   NETWORK 2
   TITLE = Schrittkette in Grundstellung (Erweitern)
      #sq.inHome := #Grundstellung.X AND "FG01Actors".Gripper.inHomePos AND "FG01Actors".Plattform.inHomePos AND "FG01Actors".ReaderWindow.inHomePos;
   NETWORK 3
   TITLE = Startbedingung (Erweitern)
      #txStartCondition := "TransportGlobals".Index01.release;
   NETWORK 4
   TITLE = Schrittkette starten
      #sq.start := #sq.inHome AND NOT #sq.running AND #signals.releaseCycle AND NOT #signals.isHoming AND #txStartCondition;
      IF #sq.start THEN #sq.done := FALSE; END_IF;
   NETWORK 5
   TITLE = ReleaseCycle Timer
      // ENO of a box is taken as its EN; it also drops when the box reports an error
      #_w1 := #ERR_FLT AND #ACK_EF;
      #_w2 := #_w1 AND NOT #sstReleaseCycle.ErrorAck;   // rising edge
      #sstReleaseCycle.ErrorAck := #_w1;
      IF (#S_NO <> #sstReleaseCycle.No_LastCycle) OR #_w2 THEN
          #sstReleaseCycle.T := T#0MS;
          #sstReleaseCycle.TckPrev := #sstReleaseCycle.Tck;
          #sstReleaseCycle.No_LastCycle := #S_NO;
      END_IF;
      #sstReleaseCycle.Tck := TIME_TCK();
      #tdTckDiff := #sstReleaseCycle.Tck - #sstReleaseCycle.TckPrev;
      #sstReleaseCycle.TckPrev := #sstReleaseCycle.Tck;
      IF (0 <= #tdTckDiff) AND (#tdTckDiff <= 1000) AND #signals.releaseCycle THEN
          #sstReleaseCycle.T := #sstReleaseCycle.T + #tdTckDiff;
      END_IF;

   // sequencer 1
   INITIAL_STEP Initialschritt:   // S1, max time T#10S, warning time T#7S
              N    #sq.init
              R    #sq.inHoming
              R    #sq.running
              R    #sq.done
   END_STEP
   TRANSITION Automatikablauf FROM Initialschritt TO Grundstellung   // T1
      := NOT #signals.isHoming;
   END_TRANSITION
   TRANSITION Grundstellungsfahrt FROM Initialschritt TO "Start Grundstellungsfahrt"   // T5
      := #signals.isHoming;
   END_TRANSITION
   STEP Grundstellung:   // S2, max time T#10S, warning time T#7S
              N    #sq.isWaiting
              N    "FG01Globals".SQ1.readyForIndex
   END_STEP
   TRANSITION Freigabe FROM Grundstellung TO SK_läuft   // T2
      := #sq.inHome AND NOT #signals.autoIsStoping AND #sq.start AND NOT #sq.done AND #signals.releaseNextJog;
   END_TRANSITION
   STEP SK_läuft:   // S3, max time T#10S, warning time T#7S
              S    #sq.running
   END_STEP
   TRANSITION Trans3 FROM SK_läuft TO GripperToWork   // T3
      := "AlwaysTRUE";
   END_TRANSITION
   STEP Fertigmeldung:   // S4, max time T#10S, warning time T#7S
              R    #sq.running
              S    #sq.done
   END_STEP
   TRANSITION Fertig FROM Fertigmeldung TO Ende   // T4
      := "AlwaysTRUE";
   END_TRANSITION
   STEP "Start Grundstellungsfahrt":   // S5, max time T#10S, warning time T#7S
              S    #sq.inHoming
   END_STEP
   TRANSITION GST_Aktiv FROM "Start Grundstellungsfahrt" TO GS_GripperHome   // T6
      := "AlwaysTRUE";
   END_TRANSITION
   STEP "Fertig Grundstellungsfahrt":   // S6, max time T#10S, warning time T#7S
              R    #sq.inHoming
   END_STEP
   TRANSITION GST_Beendet FROM "Fertig Grundstellungsfahrt" TO Ende   // T7
      := "AlwaysTRUE";
   END_TRANSITION
   STEP Ende:   // S7, max time T#10S, warning time T#7S
   END_STEP
   TRANSITION Beendet FROM Ende TO Grundstellung   // T8, jump
      := "AlwaysTRUE";
   END_TRANSITION
   STEP ResetRelease:   // S8, max time T#10S, warning time T#7S
      supervision V := (#ResetRelease.U >= t#10s) AND NOT #DoneToIndexer.TT AND #signals.releaseCycle;
          S1  R    "TransportGlobals".Index01.release
   END_STEP
   TRANSITION DoneToIndexer FROM ResetRelease TO Fertigmeldung   // T9
      := true;
   END_TRANSITION
   STEP GS_GripperHome:   // S14, max time T#10S, warning time T#7S
      supervision V := #sstReleaseCycle.T >= #itMaxRuntime;
              R    "FG01Actors".Gripper.setWorkPos
              S    "FG01Actors".Gripper.setHomePos
   END_STEP
   TRANSITION GS_GripperInHome FROM GS_GripperHome TO GS_PlattformHome   // T15
      := "FG01Actors".Gripper.inHomePos;
   END_TRANSITION
   STEP GS_PlattformHome:   // S15, max time T#10S, warning time T#7S
      supervision V := #sstReleaseCycle.T >= #itMaxRuntime;
              S    "FG01Actors".Plattform.setHomePos
              R    "FG01Actors".Plattform.setWorkPos
   END_STEP
   TRANSITION GS_PlattformInHome FROM GS_PlattformHome TO GS_ReaderWindowHome   // T16
      := "FG01Actors".Plattform.inHomePos;
   END_TRANSITION
   STEP GS_ReaderWindowHome:   // S16, max time T#10S, warning time T#7S
      supervision V := #sstReleaseCycle.T >= #itMaxRuntime;
              R    "FG01Actors".ReaderWindow.setWorkPos
              S    "FG01Actors".ReaderWindow.setHomePos
   END_STEP
   TRANSITION GS_ReaderWindowInHome FROM GS_ReaderWindowHome TO "Fertig Grundstellungsfahrt"   // T17
      := "FG01Actors".ReaderWindow.inHomePos;
   END_TRANSITION
   STEP PlattformToWork:   // S17, max time T#10S, warning time T#7S
      supervision V := (#sstReleaseCycle.T >= #itMaxRuntime) OR (#PlattformToWork.X AND "FG01Actors".Plattform.inError);
              R    "FG01Actors".Plattform.setHomePos
              S    "FG01Actors".Plattform.setWorkPos
   END_STEP
   TRANSITION PlattformIsInWork FROM PlattformToWork TO JogS2   // T18
      := "FG01Actors".Plattform.inWorkPos;
   END_TRANSITION
   STEP ReaderWindowToWork:   // S18, max time T#10S, warning time T#7S
      supervision V := (#sstReleaseCycle.T >= #itMaxRuntime) OR (#ReaderWindowToWork.X AND "FG01Actors".ReaderWindow.inError);
              S    "FG01Actors".ReaderWindow.setWorkPos
              R    "FG01Actors".ReaderWindow.setHomePos
   END_STEP
   TRANSITION ReaderWindowInWork FROM ReaderWindowToWork TO JogS3   // T19
      := "FG01Actors".ReaderWindow.inWorkPos;
   END_TRANSITION
   STEP GripperToWork:   // S19, max time T#10S, warning time T#7S
      supervision V := (#sstReleaseCycle.T >= #itMaxRuntime) OR (#GripperToWork.X AND "FG01Actors".Gripper.inError AND false);
              S    "FG01Actors".Gripper.setWorkPos
              R    "FG01Actors".Gripper.setHomePos
   END_STEP
   TRANSITION GripperInWork FROM GripperToWork TO JogS1   // T20
      := "FG01Actors".Gripper.inWorkPos;
   END_TRANSITION
   STEP GripperToHome:   // S20, max time T#10S, warning time T#7S
      supervision V := (#sstReleaseCycle.T >= #itMaxRuntime) OR (#GripperToHome.X AND "FG01Actors".Gripper.inError);
              R    "FG01Actors".Gripper.setWorkPos
              S    "FG01Actors".Gripper.setHomePos
   END_STEP
   TRANSITION GripperInHome FROM GripperToHome TO ReaderWindowToHome   // T21
      := "FG01Actors".Gripper.inHomePos;
   END_TRANSITION
   STEP PlattformToHome:   // S21, max time T#10S, warning time T#7S
      supervision V := (#sstReleaseCycle.T >= #itMaxRuntime) OR (#PlattformToHome.X AND "FG01Actors".Plattform.inError);
              S    "FG01Actors".Plattform.setHomePos
              R    "FG01Actors".Plattform.setWorkPos
   END_STEP
   TRANSITION PlattformIsInWork_1 FROM PlattformToHome TO JogS5   // T22
      := "FG01Actors".Plattform.inHomePos;
   END_TRANSITION
   STEP JogS1:   // S28, max time T#10S, warning time T#7S
              N    #sq.jogDone
   END_STEP
   TRANSITION JogT1 FROM JogS1 TO PlattformToWork   // T30
      := #signals.releaseNextJog;
   END_TRANSITION
   STEP JogS2:   // S29, max time T#10S, warning time T#7S
              N    #sq.jogDone
   END_STEP
   TRANSITION JogT2 FROM JogS2 TO ReaderWindowToWork   // T31
      := #signals.releaseNextJog;
   END_TRANSITION
   STEP JogS3:   // S30, max time T#10S, warning time T#7S
              N    #sq.jogDone
   END_STEP
   TRANSITION JogT3 FROM JogS3 TO Cam   // T32
      := #signals.releaseNextJog;
   END_TRANSITION
   STEP JogS4:   // S31, max time T#10S, warning time T#7S
              N    #sq.jogDone
   END_STEP
   TRANSITION JogT4 FROM JogS4 TO PlattformToHome   // T33
      := #signals.releaseNextJog;
   END_TRANSITION
   STEP Cam:   // S32, max time T#10S, warning time T#7S
   END_STEP
   TRANSITION Trans34 FROM Cam TO JogS4   // T34
      := #Cam.T >= t#3s;
   END_TRANSITION
   STEP JogS5:   // S33, max time T#10S, warning time T#7S
              N    #sq.jogDone
   END_STEP
   TRANSITION JogT5 FROM JogS5 TO GripperToHome   // T35
      := #signals.releaseNextJog;
   END_TRANSITION
   STEP ReaderWindowToHome:   // S22, max time T#10S, warning time T#7S
      supervision V := (#sstReleaseCycle.T >= #itMaxRuntime) OR (#ReaderWindowToHome.X AND "FG01Actors".ReaderWindow.inError);
              R    "FG01Actors".ReaderWindow.setWorkPos
              S    "FG01Actors".ReaderWindow.setHomePos
   END_STEP
   TRANSITION ReaderWindowInHome FROM ReaderWindowToHome TO ResetRelease   // T23
      := "FG01Actors".ReaderWindow.inHomePos;
   END_TRANSITION

   // permanent post-instructions
   NETWORK 1
   TITLE = Störungssignal weitergeben
      #sq.error := #ERR_FLT;
   NETWORK 2
   TITLE = Ablauf ist aktiv
      #qxIsActive := #sq.running;
   NETWORK 3
   TITLE = steht in Grundstellung
      #qxIsInHome := #sq.inHome AND NOT #sq.running;
END_FUNCTION_BLOCK

FUNCTION "FG01StepSequences" : Void   // FC1110, FBD
TITLE = Schrittkettensteuerung
{ S7_Optimized_Access := 'TRUE' }
VERSION : 0.1
// Ersteller: Andreas Fast Automation
// E-Mail: automation@fast-andreas.de
// 
// Projekt dient zu Demonstrationszwecken und frei genutzt werden.
// 
// Bausteinbeschreibung:
   VAR_IN_OUT
      station : "typeStation";
   END_VAR
   VAR_TEMP
      tempInit : Bool;
      tempAck : Bool;
      tempSwAuto : Bool;
      tempSwMan : Bool;
      tempSwTap : Bool;
      tempPush : Bool;
   END_VAR
BEGIN

REGION Network 1: Graph Parameter
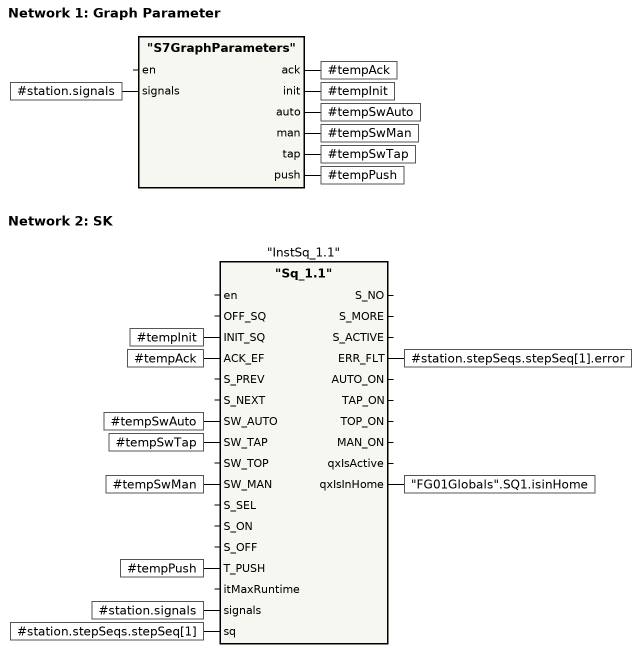
   "S7GraphParameters"(signals := #station.signals,
                       ack => #tempAck,
                       init => #tempInit,
                       auto => #tempSwAuto,
                       man => #tempSwMan,
                       tap => #tempSwTap,
                       push => #tempPush);
END_REGION

REGION Network 2: SK
   "InstSq_1.1"(INIT_SQ := #tempInit,   // "Sq_1.1"
                ACK_EF := #tempAck,
                SW_AUTO := #tempSwAuto,
                SW_TAP := #tempSwTap,
                SW_MAN := #tempSwMan,
                T_PUSH := #tempPush,
                signals := #station.signals,
                sq := #station.stepSeqs.stepSeq[1],
                ERR_FLT => #station.stepSeqs.stepSeq[1].error,
                qxIsInHome => "FG01Globals".SQ1.isinHome);
END_REGION
END_FUNCTION

// folder: 2. Machine/02_FG02

FUNCTION_BLOCK "FG02Control"   // FB1200, FBD
TITLE = Station 2 Hauptaufruf
{ S7_Optimized_Access := 'TRUE' }
VERSION : 0.1
// Ersteller: Andreas Fast Automation
// E-Mail: automation@fast-andreas.de
// 
// Projekt dient zu Demonstrationszwecken und frei genutzt werden.
// 
// Bausteinbeschreibung:
   VAR_INPUT
      stationNo : Int := 2;   // Stationsnummer
   END_VAR
   VAR_IN_OUT
      machine : "typeMachine";
      station : "typeStation";
      manualMovement : "typeManualMovements";
      plcErrMsg : "typePlcErrMsg";
      hmiErrMsg : "typeHmiErrMsg";
   END_VAR
   VAR
      instStationControl : "StationControl";
      instActorControl : "FG02ActorControl";
   END_VAR
BEGIN

REGION Network 1: Stationssteuerung
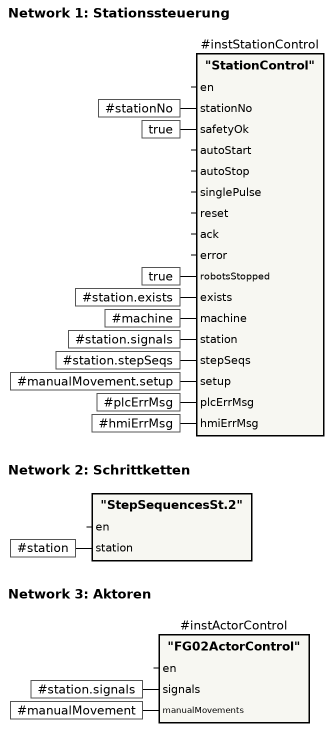
   #instStationControl(stationNo := #stationNo,   // "StationControl"
                       safetyOk := true,
                       robotsStopped := true,
                       exists := #station.exists,
                       machine := #machine,
                       station := #station.signals,
                       stepSeqs := #station.stepSeqs,
                       setup := #manualMovement.setup,
                       plcErrMsg := #plcErrMsg,
                       hmiErrMsg := #hmiErrMsg);
END_REGION

REGION Network 2: Schrittketten
   "StepSequencesSt.2"(station := #station);
END_REGION

REGION Network 3: Aktoren
   #instActorControl(signals := #station.signals, manualMovements := #manualMovement);   // "FG02ActorControl"
END_REGION
END_FUNCTION_BLOCK

FUNCTION_BLOCK "FG02ActorControl"   // FB1202, FBD
TITLE = Aktoransteuerung
{ S7_Optimized_Access := 'TRUE' }
VERSION : 0.1
// Ersteller: Andreas Fast Automation
// E-Mail: automation@fast-andreas.de
// 
// Projekt dient zu Demonstrationszwecken und frei genutzt werden.
// 
// Bausteinbeschreibung:
   VAR_IN_OUT
      signals : "typeStationSignals";
      manualMovements : "typeManualMovements";
   END_VAR
   VAR
      instActorReserved1 : "Actor_Reserved";
      instActorReserved2 : "Actor_Reserved";
      instActorReserved3 : "Actor_Reserved";
      instActorReserved4 : "Actor_Reserved";
   END_VAR
BEGIN

REGION Network 1: Reserved
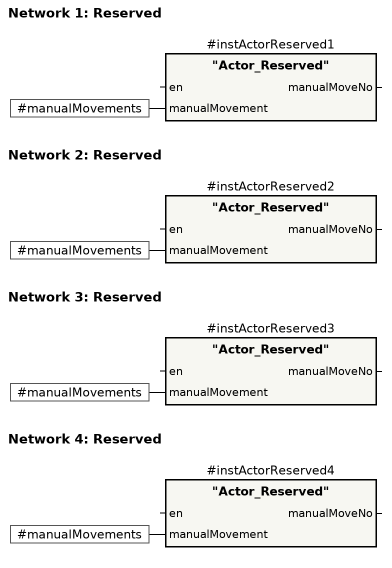
   #instActorReserved1(manualMovement := #manualMovements);   // "Actor_Reserved"
END_REGION

REGION Network 2: Reserved
   #instActorReserved2(manualMovement := #manualMovements);   // "Actor_Reserved"
END_REGION

REGION Network 3: Reserved
   #instActorReserved3(manualMovement := #manualMovements);   // "Actor_Reserved"
END_REGION

REGION Network 4: Reserved
   #instActorReserved4(manualMovement := #manualMovements);   // "Actor_Reserved"
END_REGION
END_FUNCTION_BLOCK

// folder: 2. Machine/02_FG02/Stepsequences

FUNCTION_BLOCK "Sq_2.1"   // FB1211, GRAPH_PLUS
{ S7_Optimized_Access := 'TRUE' }
VERSION : 0.1
   VAR_INPUT
      OFF_SQ : Bool := false;   // Kette ausschalten
      INIT_SQ : Bool := false;   // Kette in Initialzustand versetzen
      ACK_EF : Bool := false;   // Alle Fehler und Störungen quittieren
      S_PREV : Bool := false;   // Vorherigen Schritt am Parameter S_NO ausgeben
      S_NEXT : Bool := false;   // Nächsten Schritt am Parameter S_NO anzeigen
      SW_AUTO : Bool := false;   // Automatischer Betrieb
      SW_TAP : Bool := false;   // Halbautomatisch/Weiterschalten mit Transition
      SW_TOP : Bool := false;   // Halbautomatisch/Ignoriere Transition
      SW_MAN : Bool := false;   // Handbetrieb
      S_SEL : Int := 0;   // Schritt auswählen, der an S_NO ausgegeben werden soll
      S_ON : Bool := false;   // Schritt aktivieren, der an Parameter S_NO anliegt
      S_OFF : Bool := false;   // Schritt deaktivieren, der an Parameter S_NO anliegt
      T_PUSH : Bool := false;   // Schaltfreigabe für Transition im halbautomatischen Betrieb
      itMaxRuntime : Time := t#10s;   // Maximale Laufzeit für diesen Prozess
   END_VAR
   VAR_OUTPUT
      S_NO : Int := 0;   // Schrittnummer
      S_MORE : Bool := false;   // Weitere Schritte sind vorhanden und können in S_NO angezeigt werden.
      S_ACTIVE : Bool := false;   // Schritt, der an Parameter S_NO angezeigt wird, ist aktiv
      ERR_FLT : Bool := false;   // Sammelfehler Interlock oder Supervision
      AUTO_ON : Bool := false;   // Automatischer Betrieb eingeschaltet
      TAP_ON : Bool := false;   // Halbautomatischer Betrieb/Schritt mit Transition eingeschaltet
      TOP_ON : Bool := false;   // Halbautomatischer Betrieb/Ignoriere Transition eingeschaltet
      MAN_ON : Bool := false;   // Handbetrieb eingeschaltet
      qxIsActive : Bool;   // Schrittkette läuft
      qxIsInHome : Bool;   // steht in Grundstellung
   END_VAR
   VAR_IN_OUT
      signals : "typeStationSignals";   // Stationssteuersignale
      sq : "typeStepSequence";   // Schrittkettensteuersignale
   END_VAR
   VAR
      sstReleaseCycle : Struct
         ErrorAck : Bool;
         No_LastCycle : Int;
         T : Time;   // Aktive Zeit des ReleaseCycle
         Tck : Time;
         TckPrev : Time;
      END_STRUCT;
      HMI_INFO : Array[0..8] of UInt;
      IF_PAR : G7_IfParPlus_V6;
      RT_DATA : G7_RTDataPlus_V6;   // Interner Datenbereich
      Automatikablauf : G7_TransitionPlus_V6;   // Transitionsstruktur
      Freigabe : G7_TransitionPlus_V6;   // Transitionsstruktur
      GreiferLeer : G7_TransitionPlus_V6;   // Transitionsstruktur
      Fertig : G7_TransitionPlus_V6;   // Transitionsstruktur
      Grundstellungsfahrt : G7_TransitionPlus_V6;   // Transitionsstruktur
      GST_Aktiv : G7_TransitionPlus_V6;   // Transitionsstruktur
      GST_Beendet : G7_TransitionPlus_V6;   // Transitionsstruktur
      Beendet : G7_TransitionPlus_V6;   // Transitionsstruktur
      DoneToIndexer : G7_TransitionPlus_V6;   // Transitionsstruktur / Transition structure
      SomethingIsDone : G7_TransitionPlus_V6;   // Transitionsstruktur / Transition structure
      Initialschritt : G7_StepPlus_V6;   // Schrittstruktur
      Grundstellung : G7_StepPlus_V6;   // Schrittstruktur
      SK_läuft : G7_StepPlus_V6;   // Schrittstruktur
      Fertigmeldung : G7_StepPlus_V6;   // Schrittstruktur
      "Start Grundstellungsfahrt" : G7_StepPlus_V6;   // Schrittstruktur
      "Fertig Grundstellungsfahrt" : G7_StepPlus_V6;   // Schrittstruktur
      Ende : G7_StepPlus_V6;   // Schrittstruktur
      ResetRelease : G7_StepPlus_V6;   // Schrittstruktur / Step structure
      DoingSomething : G7_StepPlus_V6;   // Schrittstruktur / Step structure
      SINI : Array[0..1] of USInt;
      LSTT : Array[0..9] of USInt;
      ATAJ : Array[0..9] of USInt;
      ATAB : Array[0..9] of USInt;
      PSTT : Array[0..9] of USInt;
      NSTT : Array[0..9] of USInt;
      ASSJ : Array[0..8] of USInt;
      ASSB : Array[0..8] of USInt;
      PTTS : Array[0..8] of USInt;
      NTTS : Array[0..8] of USInt;
      SW_SQTS : Array[0..8] of USInt;
      SWITCH : Array[0..1] of USInt;
      TVX : Array[0..3] of USInt;
      TTX : Array[0..3] of USInt;
      TSX : Array[0..1] of USInt;
      S00X : Array[0..1] of USInt;
      SOFFX : Array[0..1] of USInt;
      SONX : Array[0..1] of USInt;
      SAX : Array[0..1] of USInt;
      SERRX : Array[0..9] of USInt;
      SMX : Array[0..9] of USInt;
      S0X : Array[0..9] of USInt;
      S1X : Array[0..9] of USInt;
      IL_ALARM_INST : Diag_Alarm;
      SUP_ALARM_INST : Diag_Alarm;
      STEP_TIME_ALARM_INST : Diag_Alarm;
      IEC_TIMER_INST : IEC_TIMER;
      TRANSACTION_FLAG : Bool := false;
   END_VAR
   VAR_TEMP
      txStartCondition : Bool;
      tdTckDiff : DInt;
   END_VAR
   VAR_TEMP   // added for the SCL form of the ladder/FBD networks
      _w1 : Bool;
   END_VAR
   // SINI[0] := 2;
   // LSTT[0] := 255;
   // LSTT[1] := 255;
   // LSTT[2] := 255;
   // LSTT[3] := 255;
   // LSTT[4] := 255;
   // LSTT[5] := 255;
   // LSTT[6] := 255;
   // LSTT[7] := 1;
   // ATAJ[1] := 1;
   // ATAJ[2] := 2;
   // ATAJ[3] := 6;
   // ATAJ[4] := 4;
   // ATAJ[5] := 5;
   // ATAJ[6] := 3;
   // ATAJ[7] := 7;
   // ATAB[0] := 4;
   // ATAB[1] := 1;
   // ATAB[2] := 2;
   // ATAB[3] := 3;
   // ATAB[5] := 5;
   // ATAB[6] := 6;
   // ATAB[7] := 7;
   // PSTT[1] := 1;
   // PSTT[2] := 2;
   // PSTT[3] := 3;
   // PSTT[5] := 4;
   // PSTT[6] := 5;
   // PSTT[7] := 6;
   // NSTT[0] := 1;
   // NSTT[1] := 2;
   // NSTT[2] := 8;
   // NSTT[3] := 6;
   // NSTT[4] := 4;
   // NSTT[5] := 5;
   // NSTT[6] := 6;
   // NSTT[7] := 1;
   // ASSJ[1] := 1;
   // ASSJ[2] := 2;
   // ASSJ[3] := 3;
   // ASSJ[4] := 4;
   // ASSJ[5] := 5;
   // ASSJ[6] := 6;
   // ASSB[1] := 1;
   // ASSB[2] := 2;
   // ASSB[3] := 3;
   // ASSB[4] := 4;
   // ASSB[5] := 5;
   // ASSB[6] := 6;
   // PTTS[0] := 255;
   // PTTS[2] := 1;
   // PTTS[3] := 8;
   // PTTS[4] := 4;
   // PTTS[5] := 5;
   // PTTS[6] := 3;
   // NTTS[1] := 1;
   // NTTS[2] := 2;
   // NTTS[3] := 3;
   // NTTS[4] := 5;
   // NTTS[5] := 6;
   // NTTS[6] := 7;
   // SW_SQTS[1] := 1;
   // SW_SQTS[2] := 1;
   // SW_SQTS[3] := 1;
   // SW_SQTS[4] := 2;
   // SW_SQTS[5] := 2;
   // SW_SQTS[6] := 3;
   // TVX[0] := 16#1;
   // TTX[0] := 16#1;
   // TSX[0] := 16#1;
   // S00X[0] := 16#1;
   // SOFFX[0] := 16#1;
   // SONX[0] := 16#1;
   // SAX[0] := 16#1;
   // SERRX[0] := 16#1;
   // SMX[0] := 16#1;
   // S0X[0] := 16#1;
   // S1X[0] := 16#1;
   // LSTT[8] := 255;
   // ATAJ[8] := 8;
   // ATAB[8] := 8;
   // PSTT[8] := 7;
   // NSTT[8] := 3;
   // ASSJ[7] := 7;
   // ASSB[7] := 7;
   // PTTS[7] := 9;
   // NTTS[7] := 8;
   // SW_SQTS[7] := 1;
   // LSTT[9] := 255;
   // ATAJ[9] := 9;
   // ATAB[9] := 9;
   // PSTT[9] := 8;
   // NSTT[9] := 7;
   // ASSJ[8] := 8;
   // ASSB[8] := 8;
   // PTTS[8] := 2;
   // NTTS[8] := 9;
   // SW_SQTS[8] := 1;
BEGIN
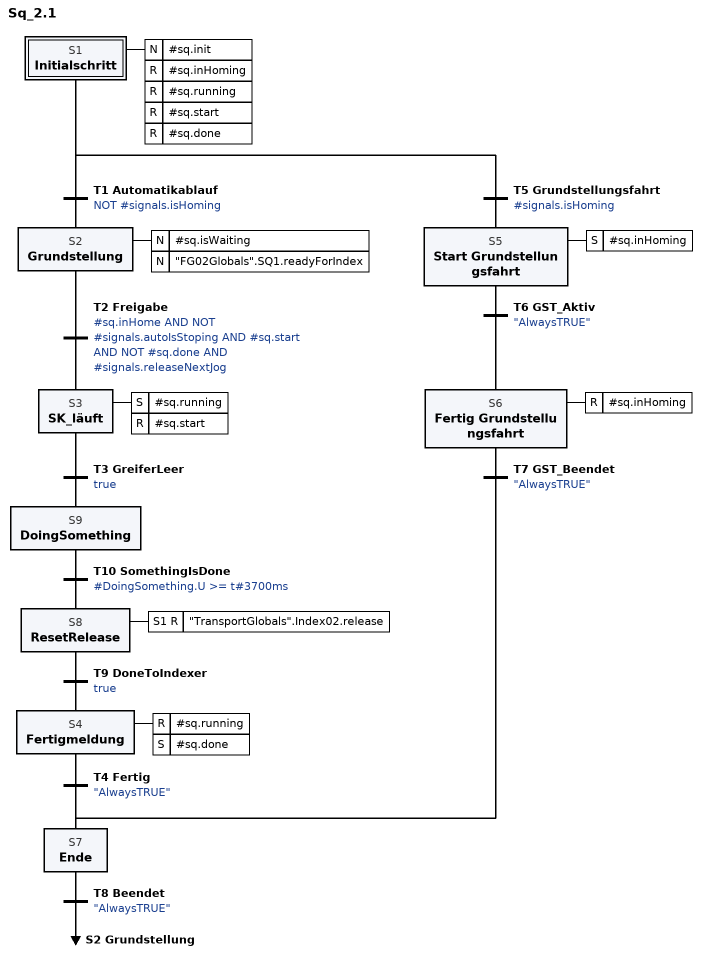
   // permanent pre-instructions
   NETWORK 1
   TITLE = Schrittkette verfügbar
      #sq.exists := true;
   NETWORK 2
   TITLE = Schrittkette in Grundstellung
      #sq.inHome := #Grundstellung.X;
   NETWORK 3
   TITLE = Startbedingung (Erweitern)
      #txStartCondition := "TransportGlobals".Index02.release;
   NETWORK 4
   TITLE = Schrittkette starten
      IF #sq.inHome AND NOT #sq.running AND #signals.releaseCycle AND NOT #signals.isHoming AND #txStartCondition THEN
          #sq.start := TRUE;
          #sq.done := FALSE;
      END_IF;
   NETWORK 5
   TITLE = ReleaseCycle Timer
      // ENO of a box is taken as its EN; it also drops when the box reports an error
      #_w1 := NOT #ERR_FLT AND #sstReleaseCycle.ErrorAck;   // falling edge
      #sstReleaseCycle.ErrorAck := #ERR_FLT;
      IF (#S_NO <> #sstReleaseCycle.No_LastCycle) OR #_w1 THEN
          #sstReleaseCycle.T := T#0MS;
          #sstReleaseCycle.TckPrev := #sstReleaseCycle.Tck;
          #sstReleaseCycle.No_LastCycle := #S_NO;
      END_IF;
      #sstReleaseCycle.Tck := TIME_TCK();
      #tdTckDiff := #sstReleaseCycle.Tck - #sstReleaseCycle.TckPrev;
      #sstReleaseCycle.TckPrev := #sstReleaseCycle.Tck;
      IF (0 <= #tdTckDiff) AND (#tdTckDiff <= 1000) AND #signals.releaseCycle THEN
          #sstReleaseCycle.T := #sstReleaseCycle.T + #tdTckDiff;
      END_IF;

   // sequencer 1
   INITIAL_STEP Initialschritt:   // S1, max time T#10S, warning time T#7S
              N    #sq.init
              R    #sq.inHoming
              R    #sq.running
              R    #sq.start
              R    #sq.done
   END_STEP
   TRANSITION Automatikablauf FROM Initialschritt TO Grundstellung   // T1
      := NOT #signals.isHoming;
   END_TRANSITION
   TRANSITION Grundstellungsfahrt FROM Initialschritt TO "Start Grundstellungsfahrt"   // T5
      := #signals.isHoming;
   END_TRANSITION
   STEP Grundstellung:   // S2, max time T#10S, warning time T#7S
      supervision V := (#Grundstellung.U > t#5S) AND NOT #sq.inHome AND #signals.releaseCycle;
              N    #sq.isWaiting
              N    "FG02Globals".SQ1.readyForIndex
   END_STEP
   TRANSITION Freigabe FROM Grundstellung TO SK_läuft   // T2
      := #sq.inHome AND NOT #signals.autoIsStoping AND #sq.start AND NOT #sq.done AND #signals.releaseNextJog;
   END_TRANSITION
   STEP SK_läuft:   // S3, max time T#10S, warning time T#7S
              S    #sq.running
              R    #sq.start
   END_STEP
   TRANSITION GreiferLeer FROM SK_läuft TO DoingSomething   // T3
      := true;
   END_TRANSITION
   STEP Fertigmeldung:   // S4, max time T#10S, warning time T#7S
              R    #sq.running
              S    #sq.done
   END_STEP
   TRANSITION Fertig FROM Fertigmeldung TO Ende   // T4
      := "AlwaysTRUE";
   END_TRANSITION
   STEP "Start Grundstellungsfahrt":   // S5, max time T#10S, warning time T#7S
              S    #sq.inHoming
   END_STEP
   TRANSITION GST_Aktiv FROM "Start Grundstellungsfahrt" TO "Fertig Grundstellungsfahrt"   // T6
      := "AlwaysTRUE";
   END_TRANSITION
   STEP "Fertig Grundstellungsfahrt":   // S6, max time T#10S, warning time T#7S
              R    #sq.inHoming
   END_STEP
   TRANSITION GST_Beendet FROM "Fertig Grundstellungsfahrt" TO Ende   // T7
      := "AlwaysTRUE";
   END_TRANSITION
   STEP Ende:   // S7, max time T#10S, warning time T#7S
   END_STEP
   TRANSITION Beendet FROM Ende TO Grundstellung   // T8, jump
      := "AlwaysTRUE";
   END_TRANSITION
   STEP DoingSomething:   // S9, max time T#10S, warning time T#7S
   END_STEP
   TRANSITION SomethingIsDone FROM DoingSomething TO ResetRelease   // T10
      := #DoingSomething.U >= t#3700ms;
   END_TRANSITION
   STEP ResetRelease:   // S8, max time T#10S, warning time T#7S
      supervision V := (#ResetRelease.U >= t#10s) AND NOT #DoneToIndexer.TT AND #signals.releaseCycle;
          S1  R    "TransportGlobals".Index02.release
   END_STEP
   TRANSITION DoneToIndexer FROM ResetRelease TO Fertigmeldung   // T9
      := true;
   END_TRANSITION

   // permanent post-instructions
   NETWORK 1
   TITLE = Störungssignal weitergeben
      #sq.error := #ERR_FLT;
   NETWORK 2
   TITLE = Ablauf ist aktiv
      #qxIsActive := #sq.running;
   NETWORK 3
   TITLE = steht in Grundstellung
      #qxIsInHome := #sq.inHome AND NOT #sq.running;
END_FUNCTION_BLOCK

FUNCTION "StepSequencesSt.2" : Void   // FC1210, FBD
TITLE = Schrittkettensteuerung
{ S7_Optimized_Access := 'TRUE' }
VERSION : 0.1
// Ersteller: Andreas Fast Automation
// E-Mail: automation@fast-andreas.de
// 
// Projekt dient zu Demonstrationszwecken und frei genutzt werden.
// 
// Bausteinbeschreibung:
   VAR_IN_OUT
      station : "typeStation";
   END_VAR
   VAR_TEMP
      tempInit : Bool;
      tempAck : Bool;
      tempAuto : Bool;
      tempMan : Bool;
      tempTap : Bool;
      tempPush : Bool;
   END_VAR
BEGIN

REGION Network 1: Graph Parameter
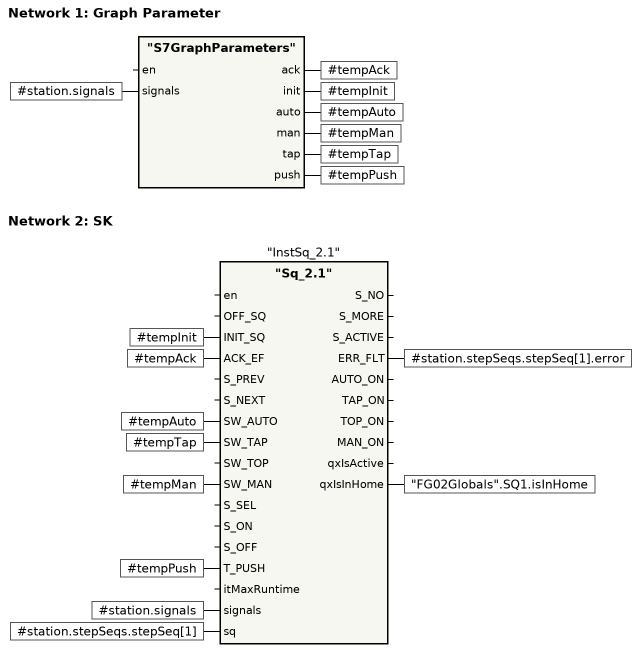
   "S7GraphParameters"(signals := #station.signals,
                       ack => #tempAck,
                       init => #tempInit,
                       auto => #tempAuto,
                       man => #tempMan,
                       tap => #tempTap,
                       push => #tempPush);
END_REGION

REGION Network 2: SK
   "InstSq_2.1"(INIT_SQ := #tempInit,   // "Sq_2.1"
                ACK_EF := #tempAck,
                SW_AUTO := #tempAuto,
                SW_TAP := #tempTap,
                SW_MAN := #tempMan,
                T_PUSH := #tempPush,
                signals := #station.signals,
                sq := #station.stepSeqs.stepSeq[1],
                ERR_FLT => #station.stepSeqs.stepSeq[1].error,
                qxIsInHome => "FG02Globals".SQ1.isInHome);
END_REGION
END_FUNCTION

// folder: 2. Machine/03_FG03

FUNCTION_BLOCK "FG03Control"   // FB1300, FBD
TITLE = Station 2 Hauptaufruf
{ S7_Optimized_Access := 'TRUE' }
VERSION : 0.1
// Ersteller: Andreas Fast Automation
// E-Mail: automation@fast-andreas.de
// 
// Projekt dient zu Demonstrationszwecken und frei genutzt werden.
// 
// Bausteinbeschreibung:
   VAR_INPUT
      stationNo : Int := 3;   // Stationsnummer
   END_VAR
   VAR_IN_OUT
      machine : "typeMachine";
      station : "typeStation";
      manualMovement : "typeManualMovements";
      plcErrMsg : "typePlcErrMsg";
      hmiErrMsg : "typeHmiErrMsg";
   END_VAR
   VAR
      instStationControl : "StationControl";
      instActorControl : "FG03ActorControl";
   END_VAR
BEGIN

REGION Network 1: Stationssteuerung
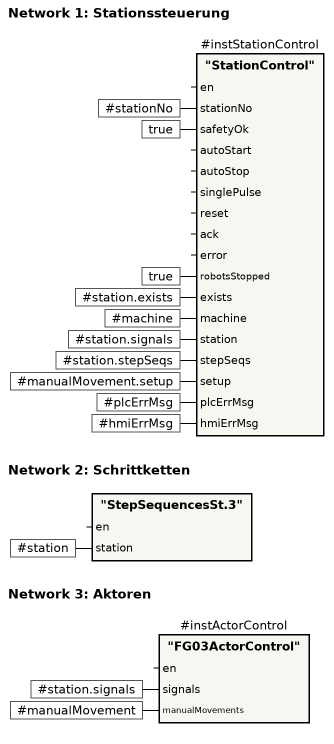
   #instStationControl(stationNo := #stationNo,   // "StationControl"
                       safetyOk := true,
                       robotsStopped := true,
                       exists := #station.exists,
                       machine := #machine,
                       station := #station.signals,
                       stepSeqs := #station.stepSeqs,
                       setup := #manualMovement.setup,
                       plcErrMsg := #plcErrMsg,
                       hmiErrMsg := #hmiErrMsg);
END_REGION

REGION Network 2: Schrittketten
   "StepSequencesSt.3"(station := #station);
END_REGION

REGION Network 3: Aktoren
   #instActorControl(signals := #station.signals, manualMovements := #manualMovement);   // "FG03ActorControl"
END_REGION
END_FUNCTION_BLOCK

FUNCTION_BLOCK "FG03ActorControl"   // FB1302, FBD
TITLE = Aktoransteuerung
{ S7_Optimized_Access := 'TRUE' }
VERSION : 0.1
// Ersteller: Andreas Fast Automation
// E-Mail: automation@fast-andreas.de
// 
// Projekt dient zu Demonstrationszwecken und frei genutzt werden.
// 
// Bausteinbeschreibung:
   VAR_IN_OUT
      signals : "typeStationSignals";
      manualMovements : "typeManualMovements";
   END_VAR
   VAR
      instActorReserved1 : "Actor_Reserved";
      instActorReserved2 : "Actor_Reserved";
      instActorReserved3 : "Actor_Reserved";
      instActorReserved4 : "Actor_Reserved";
      sinstAxisR1 : "Cylinder_2Out2In";
      sinstAxisX1 : "Cylinder_2Out2In";
      sinstAxisY1 : "Cylinder_2Out2In";
      sinstAxisX2 : "Cylinder_2Out2In";
      sinstAxisY2 : "Cylinder_2Out2In";
      sinstGripper1 : "Cylinder_2Out2In";
      sinstGripper2 : "Cylinder_2Out2In";
   END_VAR
BEGIN

REGION Network 1: AxisR1
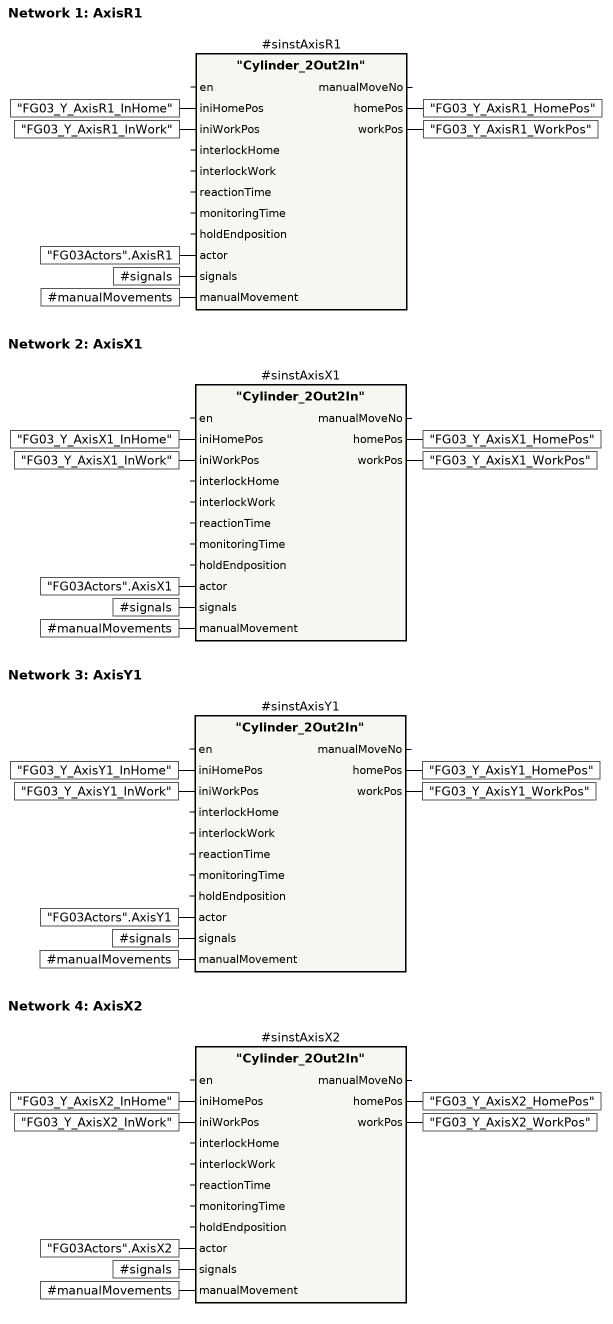
   #sinstAxisR1(iniHomePos := "FG03_Y_AxisR1_InHome",   // "Cylinder_2Out2In"
                iniWorkPos := "FG03_Y_AxisR1_InWork",
                actor := "FG03Actors".AxisR1,
                signals := #signals,
                manualMovement := #manualMovements,
                homePos => "FG03_Y_AxisR1_HomePos",
                workPos => "FG03_Y_AxisR1_WorkPos");
END_REGION

REGION Network 2: AxisX1
   #sinstAxisX1(iniHomePos := "FG03_Y_AxisX1_InHome",   // "Cylinder_2Out2In"
                iniWorkPos := "FG03_Y_AxisX1_InWork",
                actor := "FG03Actors".AxisX1,
                signals := #signals,
                manualMovement := #manualMovements,
                homePos => "FG03_Y_AxisX1_HomePos",
                workPos => "FG03_Y_AxisX1_WorkPos");
END_REGION

REGION Network 3: AxisY1
   #sinstAxisY1(iniHomePos := "FG03_Y_AxisY1_InHome",   // "Cylinder_2Out2In"
                iniWorkPos := "FG03_Y_AxisY1_InWork",
                actor := "FG03Actors".AxisY1,
                signals := #signals,
                manualMovement := #manualMovements,
                homePos => "FG03_Y_AxisY1_HomePos",
                workPos => "FG03_Y_AxisY1_WorkPos");
END_REGION

REGION Network 4: AxisX2
   #sinstAxisX2(iniHomePos := "FG03_Y_AxisX2_InHome",   // "Cylinder_2Out2In"
                iniWorkPos := "FG03_Y_AxisX2_InWork",
                actor := "FG03Actors".AxisX2,
                signals := #signals,
                manualMovement := #manualMovements,
                homePos => "FG03_Y_AxisX2_HomePos",
                workPos => "FG03_Y_AxisX2_WorkPos");
END_REGION

REGION Network 5: AxisY2
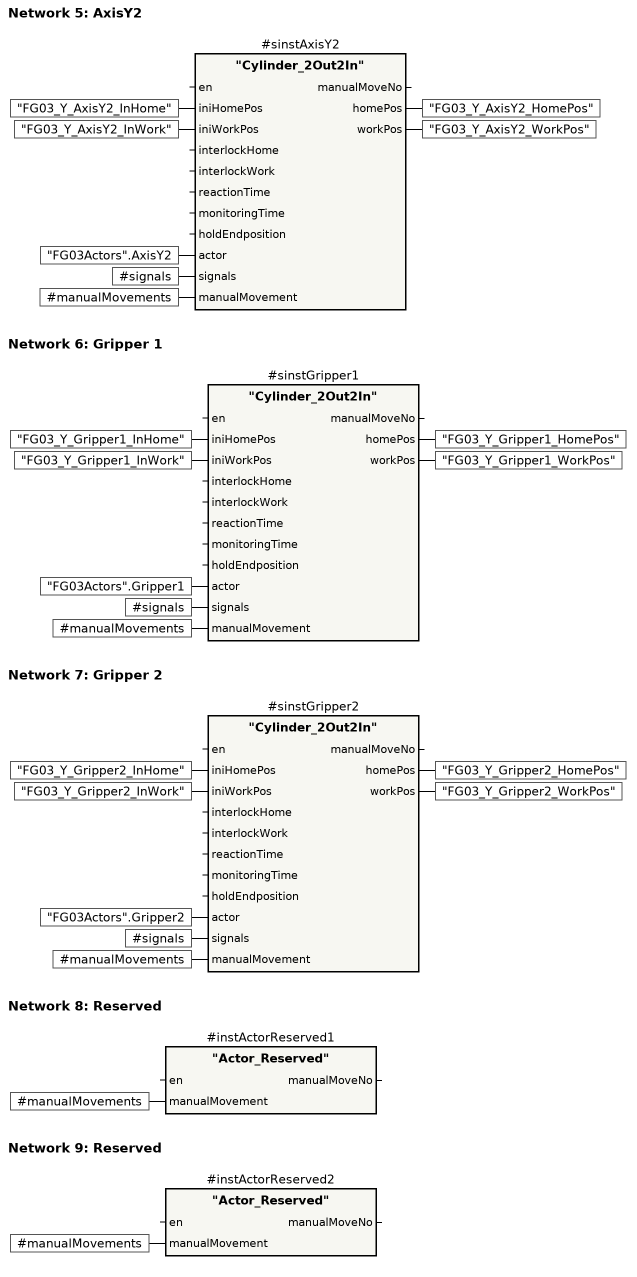
   #sinstAxisY2(iniHomePos := "FG03_Y_AxisY2_InHome",   // "Cylinder_2Out2In"
                iniWorkPos := "FG03_Y_AxisY2_InWork",
                actor := "FG03Actors".AxisY2,
                signals := #signals,
                manualMovement := #manualMovements,
                homePos => "FG03_Y_AxisY2_HomePos",
                workPos => "FG03_Y_AxisY2_WorkPos");
END_REGION

REGION Network 6: Gripper 1
   #sinstGripper1(iniHomePos := "FG03_Y_Gripper1_InHome",   // "Cylinder_2Out2In"
                  iniWorkPos := "FG03_Y_Gripper1_InWork",
                  actor := "FG03Actors".Gripper1,
                  signals := #signals,
                  manualMovement := #manualMovements,
                  homePos => "FG03_Y_Gripper1_HomePos",
                  workPos => "FG03_Y_Gripper1_WorkPos");
END_REGION

REGION Network 7: Gripper 2
   #sinstGripper2(iniHomePos := "FG03_Y_Gripper2_InHome",   // "Cylinder_2Out2In"
                  iniWorkPos := "FG03_Y_Gripper2_InWork",
                  actor := "FG03Actors".Gripper2,
                  signals := #signals,
                  manualMovement := #manualMovements,
                  homePos => "FG03_Y_Gripper2_HomePos",
                  workPos => "FG03_Y_Gripper2_WorkPos");
END_REGION

REGION Network 8: Reserved
   #instActorReserved1(manualMovement := #manualMovements);   // "Actor_Reserved"
END_REGION

REGION Network 9: Reserved
   #instActorReserved2(manualMovement := #manualMovements);   // "Actor_Reserved"
END_REGION

REGION Network 10: Reserved
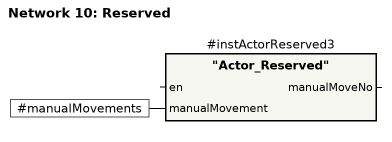
   #instActorReserved3(manualMovement := #manualMovements);   // "Actor_Reserved"
END_REGION
END_FUNCTION_BLOCK

// folder: 2. Machine/03_FG03/Stepsequences

